# B&R Automation Studio project Panasonic_LinkaPowerCP2_A2021055 (part 14)

#### Variables.var - Local variables
```iecst
VAR
	FazaNavratu : UINT := 0;
	CasSrobovania : REAL := 0.0;
	PocetCisteniSkrutkovacky : USINT := 0;
	K30_PrevodMomentu : PrevodMomentu;
	M4_PrevodMomentu : PrevodMomentu;
	M5_PrevodMomentu : PrevodMomentu;
	CasEnable_1 : TON := (0);
	CasEnable_2 : TON;
	CasEnable_3 : TON;
	CasEnable_4 : TON;
	CasResetServo_1 : TON;
	CasResetServo_2 : TON;
	CasResetServo_3 : TON;
	CasResetServo_4 : TON;
	SC_SkrutkovaciSet_K30 : SequenceControlTyp := (0);
	SC_SkrutkovaciSet_M4 : SequenceControlTyp := (0);
	SC_SkrutkovaciSet_M5 : SequenceControlTyp := (0);
	TEST : BOOL := 0;
END_VAR
```

#### AtlasCopcoKomunikacia.st
```iecst
ACTION AtlasCopcoKomunikacia:

    M4_PrevodMomentu();
    M5_PrevodMomentu();
	K30_PrevodMomentu();
	//*********************************************************Skrutkovacka M5********************************************************************************//
	//Vstupy z AtlasCopco do PLC//
    P1_Srobovanie.Skrutkovacka_M5.Stav_VysledokPotvrdeny:= P1_Srobovanie.PAR.M5_AtlasCopcoInputs[0].0;
    P1_Srobovanie.Skrutkovacka_M5.Stav_EmergencyStop:= P1_Srobovanie.PAR.M5_AtlasCopcoInputs[0].1;
    P1_Srobovanie.Skrutkovacka_M5.Stav_READY_to_START:= P1_Srobovanie.PAR.M5_AtlasCopcoInputs[0].2;
    P1_Srobovanie.Skrutkovacka_M5.Stav_MANUAL:= P1_Srobovanie.PAR.M5_AtlasCopcoInputs[0].3;
    P1_Srobovanie.Skrutkovacka_M5.Stav_UtahovanieUkoncene:= P1_Srobovanie.PAR.M5_AtlasCopcoInputs[0].4;
    P1_Srobovanie.Skrutkovacka_M5.Stav_VysledokUtahovania_NG:= P1_Srobovanie.PAR.M5_AtlasCopcoInputs[0].5;
    P1_Srobovanie.Skrutkovacka_M5.Stav_VysledokUtahovania_OK:= P1_Srobovanie.PAR.M5_AtlasCopcoInputs[0].6;
    P1_Srobovanie.Skrutkovacka_M5.Stav_SmerOtacania_VPRED:= P1_Srobovanie.PAR.M5_AtlasCopcoInputs[0].7;
    P1_Srobovanie.Skrutkovacka_M5.Stav_BUSY:= P1_Srobovanie.PAR.M5_AtlasCopcoInputs[0].8;
    P1_Srobovanie.Skrutkovacka_M5.Stav_ControlerSwitch_ON:= P1_Srobovanie.PAR.M5_AtlasCopcoInputs[0].9;
    P1_Srobovanie.Skrutkovacka_M5.Stav_Station_READY:= P1_Srobovanie.PAR.M5_AtlasCopcoInputs[0].10;
    P1_Srobovanie.Skrutkovacka_M5.Stav_NastrojPripojeny:= P1_Srobovanie.PAR.M5_AtlasCopcoInputs[0].11;
    P1_Srobovanie.Skrutkovacka_M5.Stav_NastrojUtahuje:= P1_Srobovanie.PAR.M5_AtlasCopcoInputs[0].12;

    //Výstupy z PLC do AtlasCopco//
    P1_Srobovanie.PAR.M5_AtlasCopcoOutputs[0].0:= P1_Srobovanie.Skrutkovacka_M5.RESET_Poruchy;
    P1_Srobovanie.PAR.M5_AtlasCopcoOutputs[0].1:= P1_Srobovanie.Skrutkovacka_M5.RESET_Vysledkov;
    P1_Srobovanie.PAR.M5_AtlasCopcoOutputs[0].2:= P1_Srobovanie.Skrutkovacka_M5.START_Skrutkovania;
    P1_Srobovanie.PAR.M5_AtlasCopcoOutputs[0].3:= P1_Srobovanie.Skrutkovacka_M5.START_Utahovania;

    //Číslo zadaného programu//
    P1_Srobovanie.PAR.M5_AtlasCopcoOutputs[0].16:= P1_Srobovanie.Skrutkovacka_M5.CisloZadanehoProgramu.0;
    P1_Srobovanie.PAR.M5_AtlasCopcoOutputs[0].17:= P1_Srobovanie.Skrutkovacka_M5.CisloZadanehoProgramu.1;
    P1_Srobovanie.PAR.M5_AtlasCopcoOutputs[0].18:= P1_Srobovanie.Skrutkovacka_M5.CisloZadanehoProgramu.2;
    P1_Srobovanie.PAR.M5_AtlasCopcoOutputs[0].19:= P1_Srobovanie.Skrutkovacka_M5.CisloZadanehoProgramu.3;
    P1_Srobovanie.PAR.M5_AtlasCopcoOutputs[0].20:= P1_Srobovanie.Skrutkovacka_M5.CisloZadanehoProgramu.4;
    P1_Srobovanie.PAR.M5_AtlasCopcoOutputs[0].21:= P1_Srobovanie.Skrutkovacka_M5.CisloZadanehoProgramu.5;
    P1_Srobovanie.PAR.M5_AtlasCopcoOutputs[0].22:= P1_Srobovanie.Skrutkovacka_M5.CisloZadanehoProgramu.6;
    P1_Srobovanie.PAR.M5_AtlasCopcoOutputs[0].23:= P1_Srobovanie.Skrutkovacka_M5.CisloZadanehoProgramu.7;

    //Číslo aktuálneho programu//
    P1_Srobovanie.Skrutkovacka_M5.Stav_CisloAktualnehoProgramu.0:= P1_Srobovanie.PAR.M5_AtlasCopcoInputs[5].8;
    P1_Srobovanie.Skrutkovacka_M5.Stav_CisloAktualnehoProgramu.1:= P1_Srobovanie.PAR.M5_AtlasCopcoInputs[5].9;
    P1_Srobovanie.Skrutkovacka_M5.Stav_CisloAktualnehoProgramu.2:= P1_Srobovanie.PAR.M5_AtlasCopcoInputs[5].10;
    P1_Srobovanie.Skrutkovacka_M5.Stav_CisloAktualnehoProgramu.3:= P1_Srobovanie.PAR.M5_AtlasCopcoInputs[5].11;
    P1_Srobovanie.Skrutkovacka_M5.Stav_CisloAktualnehoProgramu.4:= P1_Srobovanie.PAR.M5_AtlasCopcoInputs[5].12;
    P1_Srobovanie.Skrutkovacka_M5.Stav_CisloAktualnehoProgramu.5:= P1_Srobovanie.PAR.M5_AtlasCopcoInputs[5].13;
    P1_Srobovanie.Skrutkovacka_M5.Stav_CisloAktualnehoProgramu.6:= P1_Srobovanie.PAR.M5_AtlasCopcoInputs[5].14;
    P1_Srobovanie.Skrutkovacka_M5.Stav_CisloAktualnehoProgramu.7:= P1_Srobovanie.PAR.M5_AtlasCopcoInputs[5].15;

    //Program č.1 - skrutkovanie do plastu
    //Program č.2 - skrutkovanie do kovu

    //Dosiahnutý moment//
//    P1_Srobovanie.STAV.M5_DosiahnutyMoment.0:= P1_Srobovanie.PAR.M5_AtlasCopcoInputs[1].24;
//    P1_Srobovanie.STAV.M5_DosiahnutyMoment.1:= P1_Srobovanie.PAR.M5_AtlasCopcoInputs[1].25;
//    P1_Srobovanie.STAV.M5_DosiahnutyMoment.2:= P1_Srobovanie.PAR.M5_AtlasCopcoInputs[1].26;
//    P1_Srobovanie.STAV.M5_DosiahnutyMoment.3:= P1_Srobovanie.PAR.M5_AtlasCopcoInputs[1].27;
//    P1_Srobovanie.STAV.M5_DosiahnutyMoment.4:= P1_Srobovanie.PAR.M5_AtlasCopcoInputs[1].28;
//    P1_Srobovanie.STAV.M5_DosiahnutyMoment.5:= P1_Srobovanie.PAR.M5_AtlasCopcoInputs[1].29;
//    P1_Srobovanie.STAV.M5_DosiahnutyMoment.6:= P1_Srobovanie.PAR.M5_AtlasCopcoInputs[1].30;
//    P1_Srobovanie.STAV.M5_DosiahnutyMoment.7:= P1_Srobovanie.PAR.M5_AtlasCopcoInputs[1].31;
//    P1_Srobovanie.STAV.M5_DosiahnutyMoment.8:= P1_Srobovanie.PAR.M5_AtlasCopcoInputs[1].16;
//    P1_Srobovanie.STAV.M5_DosiahnutyMoment.9:= P1_Srobovanie.PAR.M5_AtlasCopcoInputs[1].17;
//    P1_Srobovanie.STAV.M5_DosiahnutyMoment.10:= P1_Srobovanie.PAR.M5_AtlasCopcoInputs[1].18;
//    P1_Srobovanie.STAV.M5_DosiahnutyMoment.11:= P1_Srobovanie.PAR.M5_AtlasCopcoInputs[1].19;
//    P1_Srobovanie.STAV.M5_DosiahnutyMoment.12:= P1_Srobovanie.PAR.M5_AtlasCopcoInputs[1].20;
//    P1_Srobovanie.STAV.M5_DosiahnutyMoment.13:= P1_Srobovanie.PAR.M5_AtlasCopcoInputs[1].21;
//    P1_Srobovanie.STAV.M5_DosiahnutyMoment.14:= P1_Srobovanie.PAR.M5_AtlasCopcoInputs[1].22;
//    P1_Srobovanie.STAV.M5_DosiahnutyMoment.15:= P1_Srobovanie.PAR.M5_AtlasCopcoInputs[1].23;
//    P1_Srobovanie.STAV.M5_DosiahnutyMoment.16:= P1_Srobovanie.PAR.M5_AtlasCopcoInputs[1].8;
//    P1_Srobovanie.STAV.M5_DosiahnutyMoment.17:= P1_Srobovanie.PAR.M5_AtlasCopcoInputs[1].9;
//    P1_Srobovanie.STAV.M5_DosiahnutyMoment.18:= P1_Srobovanie.PAR.M5_AtlasCopcoInputs[1].10;
//    P1_Srobovanie.STAV.M5_DosiahnutyMoment.19:= P1_Srobovanie.PAR.M5_AtlasCopcoInputs[1].11;
//    P1_Srobovanie.STAV.M5_DosiahnutyMoment.20:= P1_Srobovanie.PAR.M5_AtlasCopcoInputs[1].12;
//    P1_Srobovanie.STAV.M5_DosiahnutyMoment.21:= P1_Srobovanie.PAR.M5_AtlasCopcoInputs[1].13;
//    P1_Srobovanie.STAV.M5_DosiahnutyMoment.22:= P1_Srobovanie.PAR.M5_AtlasCopcoInputs[1].14;
//    P1_Srobovanie.STAV.M5_DosiahnutyMoment.23:= P1_Srobovanie.PAR.M5_AtlasCopcoInputs[1].15;
//    P1_Srobovanie.STAV.M5_DosiahnutyMoment.24:= P1_Srobovanie.PAR.M5_AtlasCopcoInputs[1].0;
//    P1_Srobovanie.STAV.M5_DosiahnutyMoment.25:= P1_Srobovanie.PAR.M5_AtlasCopcoInputs[1].1;
//    P1_Srobovanie.STAV.M5_DosiahnutyMoment.26:= P1_Srobovanie.PAR.M5_AtlasCopcoInputs[1].2;
//    P1_Srobovanie.STAV.M5_DosiahnutyMoment.27:= P1_Srobovanie.PAR.M5_AtlasCopcoInputs[1].3;
//    P1_Srobovanie.STAV.M5_DosiahnutyMoment.28:= P1_Srobovanie.PAR.M5_AtlasCopcoInputs[1].4;
//    P1_Srobovanie.STAV.M5_DosiahnutyMoment.29:= P1_Srobovanie.PAR.M5_AtlasCopcoInputs[1].5;
//    P1_Srobovanie.STAV.M5_DosiahnutyMoment.30:= P1_Srobovanie.PAR.M5_AtlasCopcoInputs[1].6;
//    P1_Srobovanie.STAV.M5_DosiahnutyMoment.31:= P1_Srobovanie.PAR.M5_AtlasCopcoInputs[1].7;
//    M5_DosiahnutyMoment_REAL:= UDINT_TO_REAL(P1_Srobovanie.STAV.M5_DosiahnutyMoment);
//    IF M5_DosiahnutyMoment_REAL > 0 THEN
//        P1_Srobovanie.STAV.M5_DosiahnutyMoment_REAL:= M5_DosiahnutyMoment_REAL/100;
//    ELSE
//        P1_Srobovanie.STAV.M5_DosiahnutyMoment_REAL:= 0.0;
//    END_IF

    M5_PrevodMomentu.AtlasAktualnyMoment:=P1_Srobovanie.PAR.M5_AtlasCopcoInputs[1];
    P1_Srobovanie.STAV.M5_DosiahnutyMoment_REAL:=M5_PrevodMomentu.AktualnyMoment;

    //Moment - Tolerancia MAX//
//    P1_Srobovanie.STAV.M5_Moment_ToleranciaMAX.0:= P1_Srobovanie.PAR.M5_AtlasCopcoInputs[3].24;
//    P1_Srobovanie.STAV.M5_Moment_ToleranciaMAX.1:= P1_Srobovanie.PAR.M5_AtlasCopcoInputs[3].25;
//    P1_Srobovanie.STAV.M5_Moment_ToleranciaMAX.2:= P1_Srobovanie.PAR.M5_AtlasCopcoInputs[3].26;
//    P1_Srobovanie.STAV.M5_Moment_ToleranciaMAX.3:= P1_Srobovanie.PAR.M5_AtlasCopcoInputs[3].27;
//    P1_Srobovanie.STAV.M5_Moment_ToleranciaMAX.4:= P1_Srobovanie.PAR.M5_AtlasCopcoInputs[3].28;
//    P1_Srobovanie.STAV.M5_Moment_ToleranciaMAX.5:= P1_Srobovanie.PAR.M5_AtlasCopcoInputs[3].29;
//    P1_Srobovanie.STAV.M5_Moment_ToleranciaMAX.6:= P1_Srobovanie.PAR.M5_AtlasCopcoInputs[3].30;
//    P1_Srobovanie.STAV.M5_Moment_ToleranciaMAX.7:= P1_Srobovanie.PAR.M5_AtlasCopcoInputs[3].31;
//    P1_Srobovanie.STAV.M5_Moment_ToleranciaMAX.8:= P1_Srobovanie.PAR.M5_AtlasCopcoInputs[3].16;
//    P1_Srobovanie.STAV.M5_Moment_ToleranciaMAX.9:= P1_Srobovanie.PAR.M5_AtlasCopcoInputs[3].17;
//    P1_Srobovanie.STAV.M5_Moment_ToleranciaMAX.10:= P1_Srobovanie.PAR.M5_AtlasCopcoInputs[3].18;
//    P1_Srobovanie.STAV.M5_Moment_ToleranciaMAX.11:= P1_Srobovanie.PAR.M5_AtlasCopcoInputs[3].19;
//    P1_Srobovanie.STAV.M5_Moment_ToleranciaMAX.12:= P1_Srobovanie.PAR.M5_AtlasCopcoInputs[3].20;
//    P1_Srobovanie.STAV.M5_Moment_ToleranciaMAX.13:= P1_Srobovanie.PAR.M5_AtlasCopcoInputs[3].21;
//    P1_Srobovanie.STAV.M5_Moment_ToleranciaMAX.14:= P1_Srobovanie.PAR.M5_AtlasCopcoInputs[3].22;
//    P1_Srobovanie.STAV.M5_Moment_ToleranciaMAX.15:= P1_Srobovanie.PAR.M5_AtlasCopcoInputs[3].23;
//    P1_Srobovanie.STAV.M5_Moment_ToleranciaMAX.16:= P1_Srobovanie.PAR.M5_AtlasCopcoInputs[3].8;
//    P1_Srobovanie.STAV.M5_Moment_ToleranciaMAX.17:= P1_Srobovanie.PAR.M5_AtlasCopcoInputs[3].9;
//    P1_Srobovanie.STAV.M5_Moment_ToleranciaMAX.18:= P1_Srobovanie.PAR.M5_AtlasCopcoInputs[3].10;
//    P1_Srobovanie.STAV.M5_Moment_ToleranciaMAX.19:= P1_Srobovanie.PAR.M5_AtlasCopcoInputs[3].11;
//    P1_Srobovanie.STAV.M5_Moment_ToleranciaMAX.20:= P1_Srobovanie.PAR.M5_AtlasCopcoInputs[3].12;
//    P1_Srobovanie.STAV.M5_Moment_ToleranciaMAX.21:= P1_Srobovanie.PAR.M5_AtlasCopcoInputs[3].13;
//    P1_Srobovanie.STAV.M5_Moment_ToleranciaMAX.22:= P1_Srobovanie.PAR.M5_AtlasCopcoInputs[3].14;
//    P1_Srobovanie.STAV.M5_Moment_ToleranciaMAX.23:= P1_Srobovanie.PAR.M5_AtlasCopcoInputs[3].15;
//    P1_Srobovanie.STAV.M5_Moment_ToleranciaMAX.24:= P1_Srobovanie.PAR.M5_AtlasCopcoInputs[3].0;
//    P1_Srobovanie.STAV.M5_Moment_ToleranciaMAX.25:= P1_Srobovanie.PAR.M5_AtlasCopcoInputs[3].1;
//    P1_Srobovanie.STAV.M5_Moment_ToleranciaMAX.26:= P1_Srobovanie.PAR.M5_AtlasCopcoInputs[3].2;
//    P1_Srobovanie.STAV.M5_Moment_ToleranciaMAX.27:= P1_Srobovanie.PAR.M5_AtlasCopcoInputs[3].3;
//    P1_Srobovanie.STAV.M5_Moment_ToleranciaMAX.28:= P1_Srobovanie.PAR.M5_AtlasCopcoInputs[3].4;
//    P1_Srobovanie.STAV.M5_Moment_ToleranciaMAX.29:= P1_Srobovanie.PAR.M5_AtlasCopcoInputs[3].5;
//    P1_Srobovanie.STAV.M5_Moment_ToleranciaMAX.30:= P1_Srobovanie.PAR.M5_AtlasCopcoInputs[3].6;
//    P1_Srobovanie.STAV.M5_Moment_ToleranciaMAX.31:= P1_Srobovanie.PAR.M5_AtlasCopcoInputs[3].7;
//    M5_Moment_ToleranciaMAX_REAL:= UDINT_TO_REAL(P1_Srobovanie.STAV.M5_Moment_ToleranciaMAX);
//    IF M5_Moment_ToleranciaMAX_REAL > 0 THEN
//        P1_Srobovanie.STAV.M5_Moment_ToleranciaMAX_REAL:= M5_Moment_ToleranciaMAX_REAL/100;
//    ELSE
//        P1_Srobovanie.STAV.M5_Moment_ToleranciaMAX_REAL:= 0.0;
    //    END_IF

    M5_PrevodMomentu.AtlasMaximalnaTolerancia:=P1_Srobovanie.PAR.M5_AtlasCopcoInputs[3];
    P1_Srobovanie.STAV.M5_Moment_ToleranciaMAX_REAL:=M5_PrevodMomentu.ToleranciaMAX;

    //Moment - Tolerancia MIN//
//    P1_Srobovanie.STAV.M5_Moment_ToleranciaMIN.0:= P1_Srobovanie.PAR.M5_AtlasCopcoInputs[4].24;
//    P1_Srobovanie.STAV.M5_Moment_ToleranciaMIN.1:= P1_Srobovanie.PAR.M5_AtlasCopcoInputs[4].25;
//    P1_Srobovanie.STAV.M5_Moment_ToleranciaMIN.2:= P1_Srobovanie.PAR.M5_AtlasCopcoInputs[4].26;
//    P1_Srobovanie.STAV.M5_Moment_ToleranciaMIN.3:= P1_Srobovanie.PAR.M5_AtlasCopcoInputs[4].27;
//    P1_Srobovanie.STAV.M5_Moment_ToleranciaMIN.4:= P1_Srobovanie.PAR.M5_AtlasCopcoInputs[4].28;
//    P1_Srobovanie.STAV.M5_Moment_ToleranciaMIN.5:= P1_Srobovanie.PAR.M5_AtlasCopcoInputs[4].29;
//    P1_Srobovanie.STAV.M5_Moment_ToleranciaMIN.6:= P1_Srobovanie.PAR.M5_AtlasCopcoInputs[4].30;
//    P1_Srobovanie.STAV.M5_Moment_ToleranciaMIN.7:= P1_Srobovanie.PAR.M5_AtlasCopcoInputs[4].31;
//    P1_Srobovanie.STAV.M5_Moment_ToleranciaMIN.8:= P1_Srobovanie.PAR.M5_AtlasCopcoInputs[4].16;
//    P1_Srobovanie.STAV.M5_Moment_ToleranciaMIN.9:= P1_Srobovanie.PAR.M5_AtlasCopcoInputs[4].17;
//    P1_Srobovanie.STAV.M5_Moment_ToleranciaMIN.10:= P1_Srobovanie.PAR.M5_AtlasCopcoInputs[4].18;
//    P1_Srobovanie.STAV.M5_Moment_ToleranciaMIN.11:= P1_Srobovanie.PAR.M5_AtlasCopcoInputs[4].19;
//    P1_Srobovanie.STAV.M5_Moment_ToleranciaMIN.12:= P1_Srobovanie.PAR.M5_AtlasCopcoInputs[4].20;
//    P1_Srobovanie.STAV.M5_Moment_ToleranciaMIN.13:= P1_Srobovanie.PAR.M5_AtlasCopcoInputs[4].21;
//    P1_Srobovanie.STAV.M5_Moment_ToleranciaMIN.14:= P1_Srobovanie.PAR.M5_AtlasCopcoInputs[4].22;
//    P1_Srobovanie.STAV.M5_Moment_ToleranciaMIN.15:= P1_Srobovanie.PAR.M5_AtlasCopcoInputs[4].23;
//    P1_Srobovanie.STAV.M5_Moment_ToleranciaMIN.16:= P1_Srobovanie.PAR.M5_AtlasCopcoInputs[4].8;
//    P1_Srobovanie.STAV.M5_Moment_ToleranciaMIN.17:= P1_Srobovanie.PAR.M5_AtlasCopcoInputs[4].9;
//    P1_Srobovanie.STAV.M5_Moment_ToleranciaMIN.18:= P1_Srobovanie.PAR.M5_AtlasCopcoInputs[4].10;
//    P1_Srobovanie.STAV.M5_Moment_ToleranciaMIN.19:= P1_Srobovanie.PAR.M5_AtlasCopcoInputs[4].11;
//    P1_Srobovanie.STAV.M5_Moment_ToleranciaMIN.20:= P1_Srobovanie.PAR.M5_AtlasCopcoInputs[4].12;
//    P1_Srobovanie.STAV.M5_Moment_ToleranciaMIN.21:= P1_Srobovanie.PAR.M5_AtlasCopcoInputs[4].13;
//    P1_Srobovanie.STAV.M5_Moment_ToleranciaMIN.22:= P1_Srobovanie.PAR.M5_AtlasCopcoInputs[4].14;
//    P1_Srobovanie.STAV.M5_Moment_ToleranciaMIN.23:= P1_Srobovanie.PAR.M5_AtlasCopcoInputs[4].15;
//    P1_Srobovanie.STAV.M5_Moment_ToleranciaMIN.24:= P1_Srobovanie.PAR.M5_AtlasCopcoInputs[4].0;
//    P1_Srobovanie.STAV.M5_Moment_ToleranciaMIN.25:= P1_Srobovanie.PAR.M5_AtlasCopcoInputs[4].1;
//    P1_Srobovanie.STAV.M5_Moment_ToleranciaMIN.26:= P1_Srobovanie.PAR.M5_AtlasCopcoInputs[4].2;
//    P1_Srobovanie.STAV.M5_Moment_ToleranciaMIN.27:= P1_Srobovanie.PAR.M5_AtlasCopcoInputs[4].3;
//    P1_Srobovanie.STAV.M5_Moment_ToleranciaMIN.28:= P1_Srobovanie.PAR.M5_AtlasCopcoInputs[4].4;
//    P1_Srobovanie.STAV.M5_Moment_ToleranciaMIN.29:= P1_Srobovanie.PAR.M5_AtlasCopcoInputs[4].5;
//    P1_Srobovanie.STAV.M5_Moment_ToleranciaMIN.30:= P1_Srobovanie.PAR.M5_AtlasCopcoInputs[4].6;
//    P1_Srobovanie.STAV.M5_Moment_ToleranciaMIN.31:= P1_Srobovanie.PAR.M5_AtlasCopcoInputs[4].7;
//    M5_Moment_ToleranciaMIN_REAL:= UDINT_TO_REAL(P1_Srobovanie.STAV.M5_Moment_ToleranciaMIN);
//    IF M5_Moment_ToleranciaMIN_REAL > 0 THEN
//        P1_Srobovanie.STAV.M5_Moment_ToleranciaMIN_REAL:= M5_Moment_ToleranciaMIN_REAL /100;
//    ELSE
//        P1_Srobovanie.STAV.M5_Moment_ToleranciaMIN_REAL:= 0.0;
    //    END_IF

    M5_PrevodMomentu.AtlasMinimalnaTolerancia:=P1_Srobovanie.PAR.M5_AtlasCopcoInputs[4];
    P1_Srobovanie.STAV.M5_Moment_ToleranciaMIN_REAL:=M5_PrevodMomentu.ToleranciaMIN;

    //Dosiahnutý úhol//
    P1_Srobovanie.STAV.M5_DosiahnutyUhol.0:= P1_Srobovanie.PAR.M5_AtlasCopcoInputs[0].24;
    P1_Srobovanie.STAV.M5_DosiahnutyUhol.1:= P1_Srobovanie.PAR.M5_AtlasCopcoInputs[0].25;
    P1_Srobovanie.STAV.M5_DosiahnutyUhol.2:= P1_Srobovanie.PAR.M5_AtlasCopcoInputs[0].26;
    P1_Srobovanie.STAV.M5_DosiahnutyUhol.3:= P1_Srobovanie.PAR.M5_AtlasCopcoInputs[0].27;
    P1_Srobovanie.STAV.M5_DosiahnutyUhol.4:= P1_Srobovanie.PAR.M5_AtlasCopcoInputs[0].28;
    P1_Srobovanie.STAV.M5_DosiahnutyUhol.5:= P1_Srobovanie.PAR.M5_AtlasCopcoInputs[0].29;
    P1_Srobovanie.STAV.M5_DosiahnutyUhol.6:= P1_Srobovanie.PAR.M5_AtlasCopcoInputs[0].30;
    P1_Srobovanie.STAV.M5_DosiahnutyUhol.7:= P1_Srobovanie.PAR.M5_AtlasCopcoInputs[0].31;
    P1_Srobovanie.STAV.M5_DosiahnutyUhol.8:= P1_Srobovanie.PAR.M5_AtlasCopcoInputs[0].16;
    P1_Srobovanie.STAV.M5_DosiahnutyUhol.9:= P1_Srobovanie.PAR.M5_AtlasCopcoInputs[0].17;
    P1_Srobovanie.STAV.M5_DosiahnutyUhol.10:= P1_Srobovanie.PAR.M5_AtlasCopcoInputs[0].18;
    P1_Srobovanie.STAV.M5_DosiahnutyUhol.11:= P1_Srobovanie.PAR.M5_AtlasCopcoInputs[0].19;
    P1_Srobovanie.STAV.M5_DosiahnutyUhol.12:= P1_Srobovanie.PAR.M5_AtlasCopcoInputs[0].20;
    P1_Srobovanie.STAV.M5_DosiahnutyUhol.13:= P1_Srobovanie.PAR.M5_AtlasCopcoInputs[0].21;
    P1_Srobovanie.STAV.M5_DosiahnutyUhol.14:= P1_Srobovanie.PAR.M5_AtlasCopcoInputs[0].22;
    P1_Srobovanie.STAV.M5_DosiahnutyUhol.15:= P1_Srobovanie.PAR.M5_AtlasCopcoInputs[0].23;

    //Uhol - Tolerancia MAX//
    P1_Srobovanie.STAV.M5_Uhol_ToleranciaMAX.0:= P1_Srobovanie.PAR.M5_AtlasCopcoInputs[2].8;
    P1_Srobovanie.STAV.M5_Uhol_ToleranciaMAX.1:= P1_Srobovanie.PAR.M5_AtlasCopcoInputs[2].9;
    P1_Srobovanie.STAV.M5_Uhol_ToleranciaMAX.2:= P1_Srobovanie.PAR.M5_AtlasCopcoInputs[2].10;
    P1_Srobovanie.STAV.M5_Uhol_ToleranciaMAX.3:= P1_Srobovanie.PAR.M5_AtlasCopcoInputs[2].11;
    P1_Srobovanie.STAV.M5_Uhol_ToleranciaMAX.4:= P1_Srobovanie.PAR.M5_AtlasCopcoInputs[2].12;
    P1_Srobovanie.STAV.M5_Uhol_ToleranciaMAX.5:= P1_Srobovanie.PAR.M5_AtlasCopcoInputs[2].13;
    P1_Srobovanie.STAV.M5_Uhol_ToleranciaMAX.6:= P1_Srobovanie.PAR.M5_AtlasCopcoInputs[2].14;
    P1_Srobovanie.STAV.M5_Uhol_ToleranciaMAX.7:= P1_Srobovanie.PAR.M5_AtlasCopcoInputs[2].15;
    P1_Srobovanie.STAV.M5_Uhol_ToleranciaMAX.8:= P1_Srobovanie.PAR.M5_AtlasCopcoInputs[2].0;
    P1_Srobovanie.STAV.M5_Uhol_ToleranciaMAX.9:= P1_Srobovanie.PAR.M5_AtlasCopcoInputs[2].1;
    P1_Srobovanie.STAV.M5_Uhol_ToleranciaMAX.10:= P1_Srobovanie.PAR.M5_AtlasCopcoInputs[2].2;
    P1_Srobovanie.STAV.M5_Uhol_ToleranciaMAX.11:= P1_Srobovanie.PAR.M5_AtlasCopcoInputs[2].3;
    P1_Srobovanie.STAV.M5_Uhol_ToleranciaMAX.12:= P1_Srobovanie.PAR.M5_AtlasCopcoInputs[2].4;
    P1_Srobovanie.STAV.M5_Uhol_ToleranciaMAX.13:= P1_Srobovanie.PAR.M5_AtlasCopcoInputs[2].5;
    P1_Srobovanie.STAV.M5_Uhol_ToleranciaMAX.14:= P1_Srobovanie.PAR.M5_AtlasCopcoInputs[2].6;
    P1_Srobovanie.STAV.M5_Uhol_ToleranciaMAX.15:= P1_Srobovanie.PAR.M5_AtlasCopcoInputs[2].7;

    //Uhol - Tolerancia MIN//
    P1_Srobovanie.STAV.M5_Uhol_ToleranciaMIN.0:= P1_Srobovanie.PAR.M5_AtlasCopcoInputs[2].24;
    P1_Srobovanie.STAV.M5_Uhol_ToleranciaMIN.1:= P1_Srobovanie.PAR.M5_AtlasCopcoInputs[2].25;
    P1_Srobovanie.STAV.M5_Uhol_ToleranciaMIN.2:= P1_Srobovanie.PAR.M5_AtlasCopcoInputs[2].26;
    P1_Srobovanie.STAV.M5_Uhol_ToleranciaMIN.3:= P1_Srobovanie.PAR.M5_AtlasCopcoInputs[2].27;
    P1_Srobovanie.STAV.M5_Uhol_ToleranciaMIN.4:= P1_Srobovanie.PAR.M5_AtlasCopcoInputs[2].28;
    P1_Srobovanie.STAV.M5_Uhol_ToleranciaMIN.5:= P1_Srobovanie.PAR.M5_AtlasCopcoInputs[2].29;
    P1_Srobovanie.STAV.M5_Uhol_ToleranciaMIN.6:= P1_Srobovanie.PAR.M5_AtlasCopcoInputs[2].30;
    P1_Srobovanie.STAV.M5_Uhol_ToleranciaMIN.7:= P1_Srobovanie.PAR.M5_AtlasCopcoInputs[2].31;
    P1_Srobovanie.STAV.M5_Uhol_ToleranciaMIN.8:= P1_Srobovanie.PAR.M5_AtlasCopcoInputs[2].16;
    P1_Srobovanie.STAV.M5_Uhol_ToleranciaMIN.9:= P1_Srobovanie.PAR.M5_AtlasCopcoInputs[2].17;
    P1_Srobovanie.STAV.M5_Uhol_ToleranciaMIN.10:= P1_Srobovanie.PAR.M5_AtlasCopcoInputs[2].18;
    P1_Srobovanie.STAV.M5_Uhol_ToleranciaMIN.11:= P1_Srobovanie.PAR.M5_AtlasCopcoInputs[2].19;
    P1_Srobovanie.STAV.M5_Uhol_ToleranciaMIN.12:= P1_Srobovanie.PAR.M5_AtlasCopcoInputs[2].20;
    P1_Srobovanie.STAV.M5_Uhol_ToleranciaMIN.13:= P1_Srobovanie.PAR.M5_AtlasCopcoInputs[2].21;
    P1_Srobovanie.STAV.M5_Uhol_ToleranciaMIN.14:= P1_Srobovanie.PAR.M5_AtlasCopcoInputs[2].22;
    P1_Srobovanie.STAV.M5_Uhol_ToleranciaMIN.15:= P1_Srobovanie.PAR.M5_AtlasCopcoInputs[2].23;

    //***************************************************************Skrutkovacka M4************************************************************************************//
    //Vstupy z AtlasCopco do PLC//
    P1_Srobovanie.Skrutkovacka_M4.Stav_VysledokPotvrdeny:= P1_Srobovanie.PAR.M4_AtlasCopcoInputs[0].0;
    P1_Srobovanie.Skrutkovacka_M4.Stav_EmergencyStop:= P1_Srobovanie.PAR.M4_AtlasCopcoInputs[0].1;
    P1_Srobovanie.Skrutkovacka_M4.Stav_READY_to_START:= P1_Srobovanie.PAR.M4_AtlasCopcoInputs[0].2;
    P1_Srobovanie.Skrutkovacka_M4.Stav_MANUAL:= P1_Srobovanie.PAR.M4_AtlasCopcoInputs[0].3;
    P1_Srobovanie.Skrutkovacka_M4.Stav_UtahovanieUkoncene:= P1_Srobovanie.PAR.M4_AtlasCopcoInputs[0].4;
    P1_Srobovanie.Skrutkovacka_M4.Stav_VysledokUtahovania_NG:= P1_Srobovanie.PAR.M4_AtlasCopcoInputs[0].5;
    P1_Srobovanie.Skrutkovacka_M4.Stav_VysledokUtahovania_OK:= P1_Srobovanie.PAR.M4_AtlasCopcoInputs[0].6;
    P1_Srobovanie.Skrutkovacka_M4.Stav_SmerOtacania_VPRED:= P1_Srobovanie.PAR.M4_AtlasCopcoInputs[0].7;
    P1_Srobovanie.Skrutkovacka_M4.Stav_BUSY:= P1_Srobovanie.PAR.M4_AtlasCopcoInputs[0].8;
    P1_Srobovanie.Skrutkovacka_M4.Stav_ControlerSwitch_ON:= P1_Srobovanie.PAR.M4_AtlasCopcoInputs[0].9;
    P1_Srobovanie.Skrutkovacka_M4.Stav_Station_READY:= P1_Srobovanie.PAR.M4_AtlasCopcoInputs[0].10;
    P1_Srobovanie.Skrutkovacka_M4.Stav_NastrojPripojeny:= P1_Srobovanie.PAR.M4_AtlasCopcoInputs[0].11;
    P1_Srobovanie.Skrutkovacka_M4.Stav_NastrojUtahuje:= P1_Srobovanie.PAR.M4_AtlasCopcoInputs[0].12;

    //Výstupy z PLC do AtlasCopco//
    P1_Srobovanie.PAR.M4_AtlasCopcoOutputs[0].0:= P1_Srobovanie.Skrutkovacka_M4.RESET_Poruchy;
    P1_Srobovanie.PAR.M4_AtlasCopcoOutputs[0].1:= P1_Srobovanie.Skrutkovacka_M4.RESET_Vysledkov;
    P1_Srobovanie.PAR.M4_AtlasCopcoOutputs[0].2:= P1_Srobovanie.Skrutkovacka_M4.START_Skrutkovania;
    P1_Srobovanie.PAR.M4_AtlasCopcoOutputs[0].3:= P1_Srobovanie.Skrutkovacka_M4.START_Utahovania;

    //Dosiahnutý moment//
//    P1_Srobovanie.STAV.M4_DosiahnutyMoment.0:= P1_Srobovanie.PAR.M4_AtlasCopcoInputs[1].24;
//    P1_Srobovanie.STAV.M4_DosiahnutyMoment.1:= P1_Srobovanie.PAR.M4_AtlasCopcoInputs[1].25;
//    P1_Srobovanie.STAV.M4_DosiahnutyMoment.2:= P1_Srobovanie.PAR.M4_AtlasCopcoInputs[1].26;
//    P1_Srobovanie.STAV.M4_DosiahnutyMoment.3:= P1_Srobovanie.PAR.M4_AtlasCopcoInputs[1].27;
//    P1_Srobovanie.STAV.M4_DosiahnutyMoment.4:= P1_Srobovanie.PAR.M4_AtlasCopcoInputs[1].28;
//    P1_Srobovanie.STAV.M4_DosiahnutyMoment.5:= P1_Srobovanie.PAR.M4_AtlasCopcoInputs[1].29;
//    P1_Srobovanie.STAV.M4_DosiahnutyMoment.6:= P1_Srobovanie.PAR.M4_AtlasCopcoInputs[1].30;
//    P1_Srobovanie.STAV.M4_DosiahnutyMoment.7:= P1_Srobovanie.PAR.M4_AtlasCopcoInputs[1].31;
//    P1_Srobovanie.STAV.M4_DosiahnutyMoment.8:= P1_Srobovanie.PAR.M4_AtlasCopcoInputs[1].16;
//    P1_Srobovanie.STAV.M4_DosiahnutyMoment.9:= P1_Srobovanie.PAR.M4_AtlasCopcoInputs[1].17;
//    P1_Srobovanie.STAV.M4_DosiahnutyMoment.10:= P1_Srobovanie.PAR.M4_AtlasCopcoInputs[1].18;
//    P1_Srobovanie.STAV.M4_DosiahnutyMoment.11:= P1_Srobovanie.PAR.M4_AtlasCopcoInputs[1].19;
//    P1_Srobovanie.STAV.M4_DosiahnutyMoment.12:= P1_Srobovanie.PAR.M4_AtlasCopcoInputs[1].20;
//    P1_Srobovanie.STAV.M4_DosiahnutyMoment.13:= P1_Srobovanie.PAR.M4_AtlasCopcoInputs[1].21;
//    P1_Srobovanie.STAV.M4_DosiahnutyMoment.14:= P1_Srobovanie.PAR.M4_AtlasCopcoInputs[1].22;
//    P1_Srobovanie.STAV.M4_DosiahnutyMoment.15:= P1_Srobovanie.PAR.M4_AtlasCopcoInputs[1].23;
//    P1_Srobovanie.STAV.M4_DosiahnutyMoment.16:= P1_Srobovanie.PAR.M4_AtlasCopcoInputs[1].8;
//    P1_Srobovanie.STAV.M4_DosiahnutyMoment.17:= P1_Srobovanie.PAR.M4_AtlasCopcoInputs[1].9;
//    P1_Srobovanie.STAV.M4_DosiahnutyMoment.18:= P1_Srobovanie.PAR.M4_AtlasCopcoInputs[1].10;
//    P1_Srobovanie.STAV.M4_DosiahnutyMoment.19:= P1_Srobovanie.PAR.M4_AtlasCopcoInputs[1].11;
//    P1_Srobovanie.STAV.M4_DosiahnutyMoment.20:= P1_Srobovanie.PAR.M4_AtlasCopcoInputs[1].12;
//    P1_Srobovanie.STAV.M4_DosiahnutyMoment.21:= P1_Srobovanie.PAR.M4_AtlasCopcoInputs[1].13;
//    P1_Srobovanie.STAV.M4_DosiahnutyMoment.22:= P1_Srobovanie.PAR.M4_AtlasCopcoInputs[1].14;
//    P1_Srobovanie.STAV.M4_DosiahnutyMoment.23:= P1_Srobovanie.PAR.M4_AtlasCopcoInputs[1].15;
//    P1_Srobovanie.STAV.M4_DosiahnutyMoment.24:= P1_Srobovanie.PAR.M4_AtlasCopcoInputs[1].0;
//    P1_Srobovanie.STAV.M4_DosiahnutyMoment.25:= P1_Srobovanie.PAR.M4_AtlasCopcoInputs[1].1;
//    P1_Srobovanie.STAV.M4_DosiahnutyMoment.26:= P1_Srobovanie.PAR.M4_AtlasCopcoInputs[1].2;
//    P1_Srobovanie.STAV.M4_DosiahnutyMoment.27:= P1_Srobovanie.PAR.M4_AtlasCopcoInputs[1].3;
//    P1_Srobovanie.STAV.M4_DosiahnutyMoment.28:= P1_Srobovanie.PAR.M4_AtlasCopcoInputs[1].4;
//    P1_Srobovanie.STAV.M4_DosiahnutyMoment.29:= P1_Srobovanie.PAR.M4_AtlasCopcoInputs[1].5;
//    P1_Srobovanie.STAV.M4_DosiahnutyMoment.30:= P1_Srobovanie.PAR.M4_AtlasCopcoInputs[1].6;
//    P1_Srobovanie.STAV.M4_DosiahnutyMoment.31:= P1_Srobovanie.PAR.M4_AtlasCopcoInputs[1].7;
//    M4_DosiahnutyMoment_REAL:= UDINT_TO_REAL(P1_Srobovanie.STAV.M4_DosiahnutyMoment);
//    IF M4_DosiahnutyMoment_REAL > 0 THEN
//        P1_Srobovanie.STAV.M4_DosiahnutyMoment_REAL:= (M4_DosiahnutyMoment_REAL*0.65)/42598;
//    ELSE
//        P1_Srobovanie.STAV.M4_DosiahnutyMoment_REAL:= 0.0;
//    END_IF

    M4_PrevodMomentu.AtlasAktualnyMoment:=P1_Srobovanie.PAR.M4_AtlasCopcoInputs[1];
    P1_Srobovanie.STAV.M4_DosiahnutyMoment_REAL:=M4_PrevodMomentu.AktualnyMoment;

    (*P1_Srobovanie.STAV.M4_DosiahnutyMoment_REAL:= M4_DosiahnutyMoment_REAL/100;*)

    //Moment - Tolerancia MAX//
//    P1_Srobovanie.STAV.M4_Moment_ToleranciaMAX.0:= P1_Srobovanie.PAR.M4_AtlasCopcoInputs[3].24;
    //    P1_Srobovanie.STAV.M4_Moment_ToleranciaMAX.1:= P1_Srobovanie.PAR.M4_AtlasCopcoInputs[3].25;
//    P1_Srobovanie.STAV.M4_Moment_ToleranciaMAX.2:= P1_Srobovanie.PAR.M4_AtlasCopcoInputs[3].26;
//    P1_Srobovanie.STAV.M4_Moment_ToleranciaMAX.3:= P1_Srobovanie.PAR.M4_AtlasCopcoInputs[3].27;
//    P1_Srobovanie.STAV.M4_Moment_ToleranciaMAX.4:= P1_Srobovanie.PAR.M4_AtlasCopcoInputs[3].28;
//    P1_Srobovanie.STAV.M4_Moment_ToleranciaMAX.5:= P1_Srobovanie.PAR.M4_AtlasCopcoInputs[3].29;
//    P1_Srobovanie.STAV.M4_Moment_ToleranciaMAX.6:= P1_Srobovanie.PAR.M4_AtlasCopcoInputs[3].30;
//    P1_Srobovanie.STAV.M4_Moment_ToleranciaMAX.7:= P1_Srobovanie.PAR.M4_AtlasCopcoInputs[3].31;
//    P1_Srobovanie.STAV.M4_Moment_ToleranciaMAX.8:= P1_Srobovanie.PAR.M4_AtlasCopcoInputs[3].16;
//    P1_Srobovanie.STAV.M4_Moment_ToleranciaMAX.9:= P1_Srobovanie.PAR.M4_AtlasCopcoInputs[3].17;
//    P1_Srobovanie.STAV.M4_Moment_ToleranciaMAX.10:= P1_Srobovanie.PAR.M4_AtlasCopcoInputs[3].18;
//    P1_Srobovanie.STAV.M4_Moment_ToleranciaMAX.11:= P1_Srobovanie.PAR.M4_AtlasCopcoInputs[3].19;
//    P1_Srobovanie.STAV.M4_Moment_ToleranciaMAX.12:= P1_Srobovanie.PAR.M4_AtlasCopcoInputs[3].20;
//    P1_Srobovanie.STAV.M4_Moment_ToleranciaMAX.13:= P1_Srobovanie.PAR.M4_AtlasCopcoInputs[3].21;
//    P1_Srobovanie.STAV.M4_Moment_ToleranciaMAX.14:= P1_Srobovanie.PAR.M4_AtlasCopcoInputs[3].22;
//    P1_Srobovanie.STAV.M4_Moment_ToleranciaMAX.15:= P1_Srobovanie.PAR.M4_AtlasCopcoInputs[3].23;
//    P1_Srobovanie.STAV.M4_Moment_ToleranciaMAX.16:= P1_Srobovanie.PAR.M4_AtlasCopcoInputs[3].8;
//    P1_Srobovanie.STAV.M4_Moment_ToleranciaMAX.17:= P1_Srobovanie.PAR.M4_AtlasCopcoInputs[3].9;
//    P1_Srobovanie.STAV.M4_Moment_ToleranciaMAX.18:= P1_Srobovanie.PAR.M4_AtlasCopcoInputs[3].10;
//    P1_Srobovanie.STAV.M4_Moment_ToleranciaMAX.19:= P1_Srobovanie.PAR.M4_AtlasCopcoInputs[3].11;
//    P1_Srobovanie.STAV.M4_Moment_ToleranciaMAX.20:= P1_Srobovanie.PAR.M4_AtlasCopcoInputs[3].12;
//    P1_Srobovanie.STAV.M4_Moment_ToleranciaMAX.21:= P1_Srobovanie.PAR.M4_AtlasCopcoInputs[3].13;
//    P1_Srobovanie.STAV.M4_Moment_ToleranciaMAX.22:= P1_Srobovanie.PAR.M4_AtlasCopcoInputs[3].14;
//    P1_Srobovanie.STAV.M4_Moment_ToleranciaMAX.23:= P1_Srobovanie.PAR.M4_AtlasCopcoInputs[3].15;
//    P1_Srobovanie.STAV.M4_Moment_ToleranciaMAX.24:= P1_Srobovanie.PAR.M4_AtlasCopcoInputs[3].0;
//    P1_Srobovanie.STAV.M4_Moment_ToleranciaMAX.25:= P1_Srobovanie.PAR.M4_AtlasCopcoInputs[3].1;
//    P1_Srobovanie.STAV.M4_Moment_ToleranciaMAX.26:= P1_Srobovanie.PAR.M4_AtlasCopcoInputs[3].2;
//    P1_Srobovanie.STAV.M4_Moment_ToleranciaMAX.27:= P1_Srobovanie.PAR.M4_AtlasCopcoInputs[3].3;
//    P1_Srobovanie.STAV.M4_Moment_ToleranciaMAX.28:= P1_Srobovanie.PAR.M4_AtlasCopcoInputs[3].4;
//    P1_Srobovanie.STAV.M4_Moment_ToleranciaMAX.29:= P1_Srobovanie.PAR.M4_AtlasCopcoInputs[3].5;
//    P1_Srobovanie.STAV.M4_Moment_ToleranciaMAX.30:= P1_Srobovanie.PAR.M4_AtlasCopcoInputs[3].6;
//    P1_Srobovanie.STAV.M4_Moment_ToleranciaMAX.31:= P1_Srobovanie.PAR.M4_AtlasCopcoInputs[3].7;
//    M4_Moment_ToleranciaMAX_REAL:= UDINT_TO_REAL(P1_Srobovanie.STAV.M4_Moment_ToleranciaMAX);
//    IF M4_Moment_ToleranciaMAX_REAL > 0 THEN
//        P1_Srobovanie.STAV.M4_Moment_ToleranciaMAX_REAL:= (M4_Moment_ToleranciaMAX_REAL*0.65)/42598;
//    ELSE
//        P1_Srobovanie.STAV.M4_Moment_ToleranciaMAX_REAL:= 0.0;
//    END_IF
    (*P1_Srobovanie.STAV.M4_Moment_ToleranciaMAX_REAL:= M4_Moment_ToleranciaMAX_REAL/100;*)

    M4_PrevodMomentu.AtlasMaximalnaTolerancia:=P1_Srobovanie.PAR.M4_AtlasCopcoInputs[3];
    P1_Srobovanie.STAV.M4_Moment_ToleranciaMAX_REAL:=M4_PrevodMomentu.ToleranciaMAX;

    //Moment - Tolerancia MIN//
//    P1_Srobovanie.STAV.M4_Moment_ToleranciaMIN.0:= P1_Srobovanie.PAR.M4_AtlasCopcoInputs[4].24;
//    P1_Srobovanie.STAV.M4_Moment_ToleranciaMIN.1:= P1_Srobovanie.PAR.M4_AtlasCopcoInputs[4].25;
//    P1_Srobovanie.STAV.M4_Moment_ToleranciaMIN.2:= P1_Srobovanie.PAR.M4_AtlasCopcoInputs[4].26;
//    P1_Srobovanie.STAV.M4_Moment_ToleranciaMIN.3:= P1_Srobovanie.PAR.M4_AtlasCopcoInputs[4].27;
//    P1_Srobovanie.STAV.M4_Moment_ToleranciaMIN.4:= P1_Srobovanie.PAR.M4_AtlasCopcoInputs[4].28;
//    P1_Srobovanie.STAV.M4_Moment_ToleranciaMIN.5:= P1_Srobovanie.PAR.M4_AtlasCopcoInputs[4].29;
//    P1_Srobovanie.STAV.M4_Moment_ToleranciaMIN.6:= P1_Srobovanie.PAR.M4_AtlasCopcoInputs[4].30;
//    P1_Srobovanie.STAV.M4_Moment_ToleranciaMIN.7:= P1_Srobovanie.PAR.M4_AtlasCopcoInputs[4].31;
//    P1_Srobovanie.STAV.M4_Moment_ToleranciaMIN.8:= P1_Srobovanie.PAR.M4_AtlasCopcoInputs[4].16;
//    P1_Srobovanie.STAV.M4_Moment_ToleranciaMIN.9:= P1_Srobovanie.PAR.M4_AtlasCopcoInputs[4].17;
//    P1_Srobovanie.STAV.M4_Moment_ToleranciaMIN.10:= P1_Srobovanie.PAR.M4_AtlasCopcoInputs[4].18;
//    P1_Srobovanie.STAV.M4_Moment_ToleranciaMIN.11:= P1_Srobovanie.PAR.M4_AtlasCopcoInputs[4].19;
//    P1_Srobovanie.STAV.M4_Moment_ToleranciaMIN.12:= P1_Srobovanie.PAR.M4_AtlasCopcoInputs[4].20;
//    P1_Srobovanie.STAV.M4_Moment_ToleranciaMIN.13:= P1_Srobovanie.PAR.M4_AtlasCopcoInputs[4].21;
//    P1_Srobovanie.STAV.M4_Moment_ToleranciaMIN.14:= P1_Srobovanie.PAR.M4_AtlasCopcoInputs[4].22;
//    P1_Srobovanie.STAV.M4_Moment_ToleranciaMIN.15:= P1_Srobovanie.PAR.M4_AtlasCopcoInputs[4].23;
//    P1_Srobovanie.STAV.M4_Moment_ToleranciaMIN.16:= P1_Srobovanie.PAR.M4_AtlasCopcoInputs[4].8;
//    P1_Srobovanie.STAV.M4_Moment_ToleranciaMIN.17:= P1_Srobovanie.PAR.M4_AtlasCopcoInputs[4].9;
//    P1_Srobovanie.STAV.M4_Moment_ToleranciaMIN.18:= P1_Srobovanie.PAR.M4_AtlasCopcoInputs[4].10;
//    P1_Srobovanie.STAV.M4_Moment_ToleranciaMIN.19:= P1_Srobovanie.PAR.M4_AtlasCopcoInputs[4].11;
//    P1_Srobovanie.STAV.M4_Moment_ToleranciaMIN.20:= P1_Srobovanie.PAR.M4_AtlasCopcoInputs[4].12;
//    P1_Srobovanie.STAV.M4_Moment_ToleranciaMIN.21:= P1_Srobovanie.PAR.M4_AtlasCopcoInputs[4].13;
//    P1_Srobovanie.STAV.M4_Moment_ToleranciaMIN.22:= P1_Srobovanie.PAR.M4_AtlasCopcoInputs[4].14;
//    P1_Srobovanie.STAV.M4_Moment_ToleranciaMIN.23:= P1_Srobovanie.PAR.M4_AtlasCopcoInputs[4].15;
//    P1_Srobovanie.STAV.M4_Moment_ToleranciaMIN.24:= P1_Srobovanie.PAR.M4_AtlasCopcoInputs[4].0;
//    P1_Srobovanie.STAV.M4_Moment_ToleranciaMIN.25:= P1_Srobovanie.PAR.M4_AtlasCopcoInputs[4].1;
//    P1_Srobovanie.STAV.M4_Moment_ToleranciaMIN.26:= P1_Srobovanie.PAR.M4_AtlasCopcoInputs[4].2;
//    P1_Srobovanie.STAV.M4_Moment_ToleranciaMIN.27:= P1_Srobovanie.PAR.M4_AtlasCopcoInputs[4].3;
//    P1_Srobovanie.STAV.M4_Moment_ToleranciaMIN.28:= P1_Srobovanie.PAR.M4_AtlasCopcoInputs[4].4;
//    P1_Srobovanie.STAV.M4_Moment_ToleranciaMIN.29:= P1_Srobovanie.PAR.M4_AtlasCopcoInputs[4].5;
//    P1_Srobovanie.STAV.M4_Moment_ToleranciaMIN.30:= P1_Srobovanie.PAR.M4_AtlasCopcoInputs[4].6;
//    P1_Srobovanie.STAV.M4_Moment_ToleranciaMIN.31:= P1_Srobovanie.PAR.M4_AtlasCopcoInputs[4].7;
//    M4_Moment_ToleranciaMIN_REAL:= UDINT_TO_REAL(P1_Srobovanie.STAV.M4_Moment_ToleranciaMIN);
//    IF M4_Moment_ToleranciaMIN_REAL > 0 THEN
//        P1_Srobovanie.STAV.M4_Moment_ToleranciaMIN_REAL:= (M4_Moment_ToleranciaMIN_REAL*0.65)/42598;
//    ELSE
//        P1_Srobovanie.STAV.M4_Moment_ToleranciaMIN_REAL:= 0.0;
//    END_IF
//
//
    (*P1_Srobovanie.STAV.M4_Moment_ToleranciaMIN_REAL:= M4_Moment_ToleranciaMIN_REAL /100;*)

    M4_PrevodMomentu.AtlasMinimalnaTolerancia:=P1_Srobovanie.PAR.M4_AtlasCopcoInputs[4];
    P1_Srobovanie.STAV.M4_Moment_ToleranciaMIN_REAL:=M4_PrevodMomentu.ToleranciaMIN;

    //Dosiahnutý úhol//
    P1_Srobovanie.STAV.M4_DosiahnutyUhol.0:= P1_Srobovanie.PAR.M4_AtlasCopcoInputs[0].24;
    P1_Srobovanie.STAV.M4_DosiahnutyUhol.1:= P1_Srobovanie.PAR.M4_AtlasCopcoInputs[0].25;
    P1_Srobovanie.STAV.M4_DosiahnutyUhol.2:= P1_Srobovanie.PAR.M4_AtlasCopcoInputs[0].26;
    P1_Srobovanie.STAV.M4_DosiahnutyUhol.3:= P1_Srobovanie.PAR.M4_AtlasCopcoInputs[0].27;
    P1_Srobovanie.STAV.M4_DosiahnutyUhol.4:= P1_Srobovanie.PAR.M4_AtlasCopcoInputs[0].28;
    P1_Srobovanie.STAV.M4_DosiahnutyUhol.5:= P1_Srobovanie.PAR.M4_AtlasCopcoInputs[0].29;
    P1_Srobovanie.STAV.M4_DosiahnutyUhol.6:= P1_Srobovanie.PAR.M4_AtlasCopcoInputs[0].30;
    P1_Srobovanie.STAV.M4_DosiahnutyUhol.7:= P1_Srobovanie.PAR.M4_AtlasCopcoInputs[0].31;
    P1_Srobovanie.STAV.M4_DosiahnutyUhol.8:= P1_Srobovanie.PAR.M4_AtlasCopcoInputs[0].16;
    P1_Srobovanie.STAV.M4_DosiahnutyUhol.9:= P1_Srobovanie.PAR.M4_AtlasCopcoInputs[0].17;
    P1_Srobovanie.STAV.M4_DosiahnutyUhol.10:= P1_Srobovanie.PAR.M4_AtlasCopcoInputs[0].18;
    P1_Srobovanie.STAV.M4_DosiahnutyUhol.11:= P1_Srobovanie.PAR.M4_AtlasCopcoInputs[0].19;
    P1_Srobovanie.STAV.M4_DosiahnutyUhol.12:= P1_Srobovanie.PAR.M4_AtlasCopcoInputs[0].20;
    P1_Srobovanie.STAV.M4_DosiahnutyUhol.13:= P1_Srobovanie.PAR.M4_AtlasCopcoInputs[0].21;
    P1_Srobovanie.STAV.M4_DosiahnutyUhol.14:= P1_Srobovanie.PAR.M4_AtlasCopcoInputs[0].22;
    P1_Srobovanie.STAV.M4_DosiahnutyUhol.15:= P1_Srobovanie.PAR.M4_AtlasCopcoInputs[0].23;

    //Uhol - Tolerancia MAX//
    P1_Srobovanie.STAV.M4_Uhol_ToleranciaMAX.0:= P1_Srobovanie.PAR.M4_AtlasCopcoInputs[2].8;
    P1_Srobovanie.STAV.M4_Uhol_ToleranciaMAX.1:= P1_Srobovanie.PAR.M4_AtlasCopcoInputs[2].9;
    P1_Srobovanie.STAV.M4_Uhol_ToleranciaMAX.2:= P1_Srobovanie.PAR.M4_AtlasCopcoInputs[2].10;
    P1_Srobovanie.STAV.M4_Uhol_ToleranciaMAX.3:= P1_Srobovanie.PAR.M4_AtlasCopcoInputs[2].11;
    P1_Srobovanie.STAV.M4_Uhol_ToleranciaMAX.4:= P1_Srobovanie.PAR.M4_AtlasCopcoInputs[2].12;
    P1_Srobovanie.STAV.M4_Uhol_ToleranciaMAX.5:= P1_Srobovanie.PAR.M4_AtlasCopcoInputs[2].13;
    P1_Srobovanie.STAV.M4_Uhol_ToleranciaMAX.6:= P1_Srobovanie.PAR.M4_AtlasCopcoInputs[2].14;
    P1_Srobovanie.STAV.M4_Uhol_ToleranciaMAX.7:= P1_Srobovanie.PAR.M4_AtlasCopcoInputs[2].15;
    P1_Srobovanie.STAV.M4_Uhol_ToleranciaMAX.8:= P1_Srobovanie.PAR.M4_AtlasCopcoInputs[2].0;
    P1_Srobovanie.STAV.M4_Uhol_ToleranciaMAX.9:= P1_Srobovanie.PAR.M4_AtlasCopcoInputs[2].1;
    P1_Srobovanie.STAV.M4_Uhol_ToleranciaMAX.10:= P1_Srobovanie.PAR.M4_AtlasCopcoInputs[2].2;
    P1_Srobovanie.STAV.M4_Uhol_ToleranciaMAX.11:= P1_Srobovanie.PAR.M4_AtlasCopcoInputs[2].3;
    P1_Srobovanie.STAV.M4_Uhol_ToleranciaMAX.12:= P1_Srobovanie.PAR.M4_AtlasCopcoInputs[2].4;
    P1_Srobovanie.STAV.M4_Uhol_ToleranciaMAX.13:= P1_Srobovanie.PAR.M4_AtlasCopcoInputs[2].5;
    P1_Srobovanie.STAV.M4_Uhol_ToleranciaMAX.14:= P1_Srobovanie.PAR.M4_AtlasCopcoInputs[2].6;
    P1_Srobovanie.STAV.M4_Uhol_ToleranciaMAX.15:= P1_Srobovanie.PAR.M4_AtlasCopcoInputs[2].7;

    //Uhol - Tolerancia MIN//
    P1_Srobovanie.STAV.M4_Uhol_ToleranciaMIN.0:= P1_Srobovanie.PAR.M4_AtlasCopcoInputs[2].24;
    P1_Srobovanie.STAV.M4_Uhol_ToleranciaMIN.1:= P1_Srobovanie.PAR.M4_AtlasCopcoInputs[2].25;
    P1_Srobovanie.STAV.M4_Uhol_ToleranciaMIN.2:= P1_Srobovanie.PAR.M4_AtlasCopcoInputs[2].26;
    P1_Srobovanie.STAV.M4_Uhol_ToleranciaMIN.3:= P1_Srobovanie.PAR.M4_AtlasCopcoInputs[2].27;
    P1_Srobovanie.STAV.M4_Uhol_ToleranciaMIN.4:= P1_Srobovanie.PAR.M4_AtlasCopcoInputs[2].28;
    P1_Srobovanie.STAV.M4_Uhol_ToleranciaMIN.5:= P1_Srobovanie.PAR.M4_AtlasCopcoInputs[2].29;
    P1_Srobovanie.STAV.M4_Uhol_ToleranciaMIN.6:= P1_Srobovanie.PAR.M4_AtlasCopcoInputs[2].30;
    P1_Srobovanie.STAV.M4_Uhol_ToleranciaMIN.7:= P1_Srobovanie.PAR.M4_AtlasCopcoInputs[2].31;
    P1_Srobovanie.STAV.M4_Uhol_ToleranciaMIN.8:= P1_Srobovanie.PAR.M4_AtlasCopcoInputs[2].16;
    P1_Srobovanie.STAV.M4_Uhol_ToleranciaMIN.9:= P1_Srobovanie.PAR.M4_AtlasCopcoInputs[2].17;
    P1_Srobovanie.STAV.M4_Uhol_ToleranciaMIN.10:= P1_Srobovanie.PAR.M4_AtlasCopcoInputs[2].18;
    P1_Srobovanie.STAV.M4_Uhol_ToleranciaMIN.11:= P1_Srobovanie.PAR.M4_AtlasCopcoInputs[2].19;
    P1_Srobovanie.STAV.M4_Uhol_ToleranciaMIN.12:= P1_Srobovanie.PAR.M4_AtlasCopcoInputs[2].20;
    P1_Srobovanie.STAV.M4_Uhol_ToleranciaMIN.13:= P1_Srobovanie.PAR.M4_AtlasCopcoInputs[2].21;
    P1_Srobovanie.STAV.M4_Uhol_ToleranciaMIN.14:= P1_Srobovanie.PAR.M4_AtlasCopcoInputs[2].22;
    P1_Srobovanie.STAV.M4_Uhol_ToleranciaMIN.15:= P1_Srobovanie.PAR.M4_AtlasCopcoInputs[2].23;

    //*********************************Skrutkovacka K30*******************************************************************************//
    //Vstupy z AtlasCopco do PLC//
    P1_Srobovanie.Skrutkovacka_K30.Stav_VysledokPotvrdeny:= P1_Srobovanie.PAR.K30_AtlasCopcoInputs[0].0;
    P1_Srobovanie.Skrutkovacka_K30.Stav_EmergencyStop:= P1_Srobovanie.PAR.K30_AtlasCopcoInputs[0].1;
    P1_Srobovanie.Skrutkovacka_K30.Stav_READY_to_START:= P1_Srobovanie.PAR.K30_AtlasCopcoInputs[0].2;
    P1_Srobovanie.Skrutkovacka_K30.Stav_MANUAL:= P1_Srobovanie.PAR.K30_AtlasCopcoInputs[0].3;
    P1_Srobovanie.Skrutkovacka_K30.Stav_UtahovanieUkoncene:= P1_Srobovanie.PAR.K30_AtlasCopcoInputs[0].4;
    P1_Srobovanie.Skrutkovacka_K30.Stav_VysledokUtahovania_NG:= P1_Srobovanie.PAR.K30_AtlasCopcoInputs[0].5;
    P1_Srobovanie.Skrutkovacka_K30.Stav_VysledokUtahovania_OK:= P1_Srobovanie.PAR.K30_AtlasCopcoInputs[0].6;
    P1_Srobovanie.Skrutkovacka_K30.Stav_SmerOtacania_VPRED:= P1_Srobovanie.PAR.K30_AtlasCopcoInputs[0].7;
    P1_Srobovanie.Skrutkovacka_K30.Stav_BUSY:= P1_Srobovanie.PAR.K30_AtlasCopcoInputs[0].8; //Další byte
    P1_Srobovanie.Skrutkovacka_K30.Stav_ControlerSwitch_ON:= P1_Srobovanie.PAR.K30_AtlasCopcoInputs[0].9;
    P1_Srobovanie.Skrutkovacka_K30.Stav_Station_READY:= P1_Srobovanie.PAR.K30_AtlasCopcoInputs[0].10;
    P1_Srobovanie.Skrutkovacka_K30.Stav_NastrojPripojeny:= P1_Srobovanie.PAR.K30_AtlasCopcoInputs[0].11;
    P1_Srobovanie.Skrutkovacka_K30.Stav_NastrojUtahuje:= P1_Srobovanie.PAR.K30_AtlasCopcoInputs[0].12;

    //Výstupy z PLC do AtlasCopco//
    P1_Srobovanie.PAR.K30_AtlasCopcoOutputs[0].0:= P1_Srobovanie.Skrutkovacka_K30.RESET_Poruchy;
    P1_Srobovanie.PAR.K30_AtlasCopcoOutputs[0].1:= P1_Srobovanie.Skrutkovacka_K30.RESET_Vysledkov;
    P1_Srobovanie.PAR.K30_AtlasCopcoOutputs[0].2:= P1_Srobovanie.Skrutkovacka_K30.START_Skrutkovania;
    P1_Srobovanie.PAR.K30_AtlasCopcoOutputs[0].3:= P1_Srobovanie.Skrutkovacka_K30.START_Utahovania;

    //Dosiahnutý moment//
//    P1_Srobovanie.STAV.K30_DosiahnutyMoment.0:= P1_Srobovanie.PAR.K30_AtlasCopcoInputs[1].24;
//    P1_Srobovanie.STAV.K30_DosiahnutyMoment.1:= P1_Srobovanie.PAR.K30_AtlasCopcoInputs[1].25;
//    P1_Srobovanie.STAV.K30_DosiahnutyMoment.2:= P1_Srobovanie.PAR.K30_AtlasCopcoInputs[1].26;
//    P1_Srobovanie.STAV.K30_DosiahnutyMoment.3:= P1_Srobovanie.PAR.K30_AtlasCopcoInputs[1].27;
//    P1_Srobovanie.STAV.K30_DosiahnutyMoment.4:= P1_Srobovanie.PAR.K30_AtlasCopcoInputs[1].28;
//    P1_Srobovanie.STAV.K30_DosiahnutyMoment.5:= P1_Srobovanie.PAR.K30_AtlasCopcoInputs[1].29;
//    P1_Srobovanie.STAV.K30_DosiahnutyMoment.6:= P1_Srobovanie.PAR.K30_AtlasCopcoInputs[1].30;
//    P1_Srobovanie.STAV.K30_DosiahnutyMoment.7:= P1_Srobovanie.PAR.K30_AtlasCopcoInputs[1].31;
//    P1_Srobovanie.STAV.K30_DosiahnutyMoment.8:= P1_Srobovanie.PAR.K30_AtlasCopcoInputs[1].16;
//    P1_Srobovanie.STAV.K30_DosiahnutyMoment.9:= P1_Srobovanie.PAR.K30_AtlasCopcoInputs[1].17;
//    P1_Srobovanie.STAV.K30_DosiahnutyMoment.10:= P1_Srobovanie.PAR.K30_AtlasCopcoInputs[1].18;
//    P1_Srobovanie.STAV.K30_DosiahnutyMoment.11:= P1_Srobovanie.PAR.K30_AtlasCopcoInputs[1].19;
//    P1_Srobovanie.STAV.K30_DosiahnutyMoment.12:= P1_Srobovanie.PAR.K30_AtlasCopcoInputs[1].20;
//    P1_Srobovanie.STAV.K30_DosiahnutyMoment.13:= P1_Srobovanie.PAR.K30_AtlasCopcoInputs[1].21;
//    P1_Srobovanie.STAV.K30_DosiahnutyMoment.14:= P1_Srobovanie.PAR.K30_AtlasCopcoInputs[1].22;
//    P1_Srobovanie.STAV.K30_DosiahnutyMoment.15:= P1_Srobovanie.PAR.K30_AtlasCopcoInputs[1].23;
//    P1_Srobovanie.STAV.K30_DosiahnutyMoment.16:= P1_Srobovanie.PAR.K30_AtlasCopcoInputs[1].8;
//    P1_Srobovanie.STAV.K30_DosiahnutyMoment.17:= P1_Srobovanie.PAR.K30_AtlasCopcoInputs[1].9;
//    P1_Srobovanie.STAV.K30_DosiahnutyMoment.18:= P1_Srobovanie.PAR.K30_AtlasCopcoInputs[1].10;
//    P1_Srobovanie.STAV.K30_DosiahnutyMoment.19:= P1_Srobovanie.PAR.K30_AtlasCopcoInputs[1].11;
//    P1_Srobovanie.STAV.K30_DosiahnutyMoment.20:= P1_Srobovanie.PAR.K30_AtlasCopcoInputs[1].12;
//    P1_Srobovanie.STAV.K30_DosiahnutyMoment.21:= P1_Srobovanie.PAR.K30_AtlasCopcoInputs[1].13;
//    P1_Srobovanie.STAV.K30_DosiahnutyMoment.22:= P1_Srobovanie.PAR.K30_AtlasCopcoInputs[1].14;
//    P1_Srobovanie.STAV.K30_DosiahnutyMoment.23:= P1_Srobovanie.PAR.K30_AtlasCopcoInputs[1].15;
//    P1_Srobovanie.STAV.K30_DosiahnutyMoment.24:= P1_Srobovanie.PAR.K30_AtlasCopcoInputs[1].0;
//    P1_Srobovanie.STAV.K30_DosiahnutyMoment.25:= P1_Srobovanie.PAR.K30_AtlasCopcoInputs[1].1;
//    P1_Srobovanie.STAV.K30_DosiahnutyMoment.26:= P1_Srobovanie.PAR.K30_AtlasCopcoInputs[1].2;
//    P1_Srobovanie.STAV.K30_DosiahnutyMoment.27:= P1_Srobovanie.PAR.K30_AtlasCopcoInputs[1].3;
//    P1_Srobovanie.STAV.K30_DosiahnutyMoment.28:= P1_Srobovanie.PAR.K30_AtlasCopcoInputs[1].4;
//    P1_Srobovanie.STAV.K30_DosiahnutyMoment.29:= P1_Srobovanie.PAR.K30_AtlasCopcoInputs[1].5;
//    P1_Srobovanie.STAV.K30_DosiahnutyMoment.30:= P1_Srobovanie.PAR.K30_AtlasCopcoInputs[1].6;
//    P1_Srobovanie.STAV.K30_DosiahnutyMoment.31:= P1_Srobovanie.PAR.K30_AtlasCopcoInputs[1].7;
//    K30_DosiahnutyMoment_REAL:= UDINT_TO_REAL(P1_Srobovanie.STAV.K30_DosiahnutyMoment);
//    IF K30_DosiahnutyMoment_REAL > 0 THEN
//        P1_Srobovanie.STAV.K30_DosiahnutyMoment_REAL:= K30_DosiahnutyMoment_REAL/100;
//    ELSE
//        P1_Srobovanie.STAV.K30_DosiahnutyMoment_REAL:= 0.0;
//    END_IF

    (*P1_Srobovanie.STAV.K30_DosiahnutyMoment_REAL:= (K30_DosiahnutyMoment_REAL*0.65)/42598;*)

    K30_PrevodMomentu.AtlasAktualnyMoment:=P1_Srobovanie.PAR.K30_AtlasCopcoInputs[1];
    P1_Srobovanie.STAV.K30_DosiahnutyMoment_REAL:=K30_PrevodMomentu.AktualnyMoment;

    //Moment - Tolerancia MAX//
//    P1_Srobovanie.STAV.K30_Moment_ToleranciaMAX.0:= P1_Srobovanie.PAR.K30_AtlasCopcoInputs[3].24;
//    P1_Srobovanie.STAV.K30_Moment_ToleranciaMAX.1:= P1_Srobovanie.PAR.K30_AtlasCopcoInputs[3].25;
//    P1_Srobovanie.STAV.K30_Moment_ToleranciaMAX.2:= P1_Srobovanie.PAR.K30_AtlasCopcoInputs[3].26;
//    P1_Srobovanie.STAV.K30_Moment_ToleranciaMAX.3:= P1_Srobovanie.PAR.K30_AtlasCopcoInputs[3].27;
//    P1_Srobovanie.STAV.K30_Moment_ToleranciaMAX.4:= P1_Srobovanie.PAR.K30_AtlasCopcoInputs[3].28;
//    P1_Srobovanie.STAV.K30_Moment_ToleranciaMAX.5:= P1_Srobovanie.PAR.K30_AtlasCopcoInputs[3].29;
//    P1_Srobovanie.STAV.K30_Moment_ToleranciaMAX.6:= P1_Srobovanie.PAR.K30_AtlasCopcoInputs[3].30;
//    P1_Srobovanie.STAV.K30_Moment_ToleranciaMAX.7:= P1_Srobovanie.PAR.K30_AtlasCopcoInputs[3].31;
//    P1_Srobovanie.STAV.K30_Moment_ToleranciaMAX.8:= P1_Srobovanie.PAR.K30_AtlasCopcoInputs[3].16;
//    P1_Srobovanie.STAV.K30_Moment_ToleranciaMAX.9:= P1_Srobovanie.PAR.K30_AtlasCopcoInputs[3].17;
//    P1_Srobovanie.STAV.K30_Moment_ToleranciaMAX.10:= P1_Srobovanie.PAR.K30_AtlasCopcoInputs[3].18;
//    P1_Srobovanie.STAV.K30_Moment_ToleranciaMAX.11:= P1_Srobovanie.PAR.K30_AtlasCopcoInputs[3].19;
//    P1_Srobovanie.STAV.K30_Moment_ToleranciaMAX.12:= P1_Srobovanie.PAR.K30_AtlasCopcoInputs[3].20;
//    P1_Srobovanie.STAV.K30_Moment_ToleranciaMAX.13:= P1_Srobovanie.PAR.K30_AtlasCopcoInputs[3].21;
//    P1_Srobovanie.STAV.K30_Moment_ToleranciaMAX.14:= P1_Srobovanie.PAR.K30_AtlasCopcoInputs[3].22;
//    P1_Srobovanie.STAV.K30_Moment_ToleranciaMAX.15:= P1_Srobovanie.PAR.K30_AtlasCopcoInputs[3].23;
//    P1_Srobovanie.STAV.K30_Moment_ToleranciaMAX.16:= P1_Srobovanie.PAR.K30_AtlasCopcoInputs[3].8;
//    P1_Srobovanie.STAV.K30_Moment_ToleranciaMAX.17:= P1_Srobovanie.PAR.K30_AtlasCopcoInputs[3].9;
//    P1_Srobovanie.STAV.K30_Moment_ToleranciaMAX.18:= P1_Srobovanie.PAR.K30_AtlasCopcoInputs[3].10;
//    P1_Srobovanie.STAV.K30_Moment_ToleranciaMAX.19:= P1_Srobovanie.PAR.K30_AtlasCopcoInputs[3].11;
//    P1_Srobovanie.STAV.K30_Moment_ToleranciaMAX.20:= P1_Srobovanie.PAR.K30_AtlasCopcoInputs[3].12;
//    P1_Srobovanie.STAV.K30_Moment_ToleranciaMAX.21:= P1_Srobovanie.PAR.K30_AtlasCopcoInputs[3].13;
//    P1_Srobovanie.STAV.K30_Moment_ToleranciaMAX.22:= P1_Srobovanie.PAR.K30_AtlasCopcoInputs[3].14;
//    P1_Srobovanie.STAV.K30_Moment_ToleranciaMAX.23:= P1_Srobovanie.PAR.K30_AtlasCopcoInputs[3].15;
//    P1_Srobovanie.STAV.K30_Moment_ToleranciaMAX.24:= P1_Srobovanie.PAR.K30_AtlasCopcoInputs[3].0;
//    P1_Srobovanie.STAV.K30_Moment_ToleranciaMAX.25:= P1_Srobovanie.PAR.K30_AtlasCopcoInputs[3].1;
//    P1_Srobovanie.STAV.K30_Moment_ToleranciaMAX.26:= P1_Srobovanie.PAR.K30_AtlasCopcoInputs[3].2;
//    P1_Srobovanie.STAV.K30_Moment_ToleranciaMAX.27:= P1_Srobovanie.PAR.K30_AtlasCopcoInputs[3].3;
//    P1_Srobovanie.STAV.K30_Moment_ToleranciaMAX.28:= P1_Srobovanie.PAR.K30_AtlasCopcoInputs[3].4;
//    P1_Srobovanie.STAV.K30_Moment_ToleranciaMAX.29:= P1_Srobovanie.PAR.K30_AtlasCopcoInputs[3].5;
//    P1_Srobovanie.STAV.K30_Moment_ToleranciaMAX.30:= P1_Srobovanie.PAR.K30_AtlasCopcoInputs[3].6;
//    P1_Srobovanie.STAV.K30_Moment_ToleranciaMAX.31:= P1_Srobovanie.PAR.K30_AtlasCopcoInputs[3].7;
//    K30_Moment_ToleranciaMAX_REAL:= UDINT_TO_REAL(P1_Srobovanie.STAV.K30_Moment_ToleranciaMAX);
//    IF K30_Moment_ToleranciaMAX_REAL > 0 THEN
//       P1_Srobovanie.STAV.K30_Moment_ToleranciaMAX_REAL:= K30_Moment_ToleranciaMAX_REAL/100;
//    ELSE
//        P1_Srobovanie.STAV.K30_Moment_ToleranciaMAX_REAL:= 0.0;
//    END_IF

    (*P1_Srobovanie.STAV.K30_Moment_ToleranciaMAX_REAL:= (K30_Moment_ToleranciaMAX_REAL*0.65)/42598;*)
    K30_PrevodMomentu.AtlasMaximalnaTolerancia:=P1_Srobovanie.PAR.K30_AtlasCopcoInputs[3];
    P1_Srobovanie.STAV.K30_Moment_ToleranciaMAX_REAL:=K30_PrevodMomentu.ToleranciaMAX;

    //Moment - Tolerancia MIN//
//    P1_Srobovanie.STAV.K30_Moment_ToleranciaMIN.0:= P1_Srobovanie.PAR.K30_AtlasCopcoInputs[4].24;
//    P1_Srobovanie.STAV.K30_Moment_ToleranciaMIN.1:= P1_Srobovanie.PAR.K30_AtlasCopcoInputs[4].25;
//    P1_Srobovanie.STAV.K30_Moment_ToleranciaMIN.2:= P1_Srobovanie.PAR.K30_AtlasCopcoInputs[4].26;
//    P1_Srobovanie.STAV.K30_Moment_ToleranciaMIN.3:= P1_Srobovanie.PAR.K30_AtlasCopcoInputs[4].27;
//    P1_Srobovanie.STAV.K30_Moment_ToleranciaMIN.4:= P1_Srobovanie.PAR.K30_AtlasCopcoInputs[4].28;
//    P1_Srobovanie.STAV.K30_Moment_ToleranciaMIN.5:= P1_Srobovanie.PAR.K30_AtlasCopcoInputs[4].29;
//    P1_Srobovanie.STAV.K30_Moment_ToleranciaMIN.6:= P1_Srobovanie.PAR.K30_AtlasCopcoInputs[4].30;
//    P1_Srobovanie.STAV.K30_Moment_ToleranciaMIN.7:= P1_Srobovanie.PAR.K30_AtlasCopcoInputs[4].31;
//    P1_Srobovanie.STAV.K30_Moment_ToleranciaMIN.8:= P1_Srobovanie.PAR.K30_AtlasCopcoInputs[4].16;
//    P1_Srobovanie.STAV.K30_Moment_ToleranciaMIN.9:= P1_Srobovanie.PAR.K30_AtlasCopcoInputs[4].17;
//    P1_Srobovanie.STAV.K30_Moment_ToleranciaMIN.10:= P1_Srobovanie.PAR.K30_AtlasCopcoInputs[4].18;
//    P1_Srobovanie.STAV.K30_Moment_ToleranciaMIN.11:= P1_Srobovanie.PAR.K30_AtlasCopcoInputs[4].19;
//    P1_Srobovanie.STAV.K30_Moment_ToleranciaMIN.12:= P1_Srobovanie.PAR.K30_AtlasCopcoInputs[4].20;
//    P1_Srobovanie.STAV.K30_Moment_ToleranciaMIN.13:= P1_Srobovanie.PAR.K30_AtlasCopcoInputs[4].21;
//    P1_Srobovanie.STAV.K30_Moment_ToleranciaMIN.14:= P1_Srobovanie.PAR.K30_AtlasCopcoInputs[4].22;
//    P1_Srobovanie.STAV.K30_Moment_ToleranciaMIN.15:= P1_Srobovanie.PAR.K30_AtlasCopcoInputs[4].23;
//    P1_Srobovanie.STAV.K30_Moment_ToleranciaMIN.16:= P1_Srobovanie.PAR.K30_AtlasCopcoInputs[4].8;
//    P1_Srobovanie.STAV.K30_Moment_ToleranciaMIN.17:= P1_Srobovanie.PAR.K30_AtlasCopcoInputs[4].9;
//    P1_Srobovanie.STAV.K30_Moment_ToleranciaMIN.18:= P1_Srobovanie.PAR.K30_AtlasCopcoInputs[4].10;
//    P1_Srobovanie.STAV.K30_Moment_ToleranciaMIN.19:= P1_Srobovanie.PAR.K30_AtlasCopcoInputs[4].11;
//    P1_Srobovanie.STAV.K30_Moment_ToleranciaMIN.20:= P1_Srobovanie.PAR.K30_AtlasCopcoInputs[4].12;
//    P1_Srobovanie.STAV.K30_Moment_ToleranciaMIN.21:= P1_Srobovanie.PAR.K30_AtlasCopcoInputs[4].13;
//    P1_Srobovanie.STAV.K30_Moment_ToleranciaMIN.22:= P1_Srobovanie.PAR.K30_AtlasCopcoInputs[4].14;
//    P1_Srobovanie.STAV.K30_Moment_ToleranciaMIN.23:= P1_Srobovanie.PAR.K30_AtlasCopcoInputs[4].15;
//    P1_Srobovanie.STAV.K30_Moment_ToleranciaMIN.24:= P1_Srobovanie.PAR.K30_AtlasCopcoInputs[4].0;
//    P1_Srobovanie.STAV.K30_Moment_ToleranciaMIN.25:= P1_Srobovanie.PAR.K30_AtlasCopcoInputs[4].1;
//    P1_Srobovanie.STAV.K30_Moment_ToleranciaMIN.26:= P1_Srobovanie.PAR.K30_AtlasCopcoInputs[4].2;
//    P1_Srobovanie.STAV.K30_Moment_ToleranciaMIN.27:= P1_Srobovanie.PAR.K30_AtlasCopcoInputs[4].3;
//    P1_Srobovanie.STAV.K30_Moment_ToleranciaMIN.28:= P1_Srobovanie.PAR.K30_AtlasCopcoInputs[4].4;
//    P1_Srobovanie.STAV.K30_Moment_ToleranciaMIN.29:= P1_Srobovanie.PAR.K30_AtlasCopcoInputs[4].5;
//    P1_Srobovanie.STAV.K30_Moment_ToleranciaMIN.30:= P1_Srobovanie.PAR.K30_AtlasCopcoInputs[4].6;
//    P1_Srobovanie.STAV.K30_Moment_ToleranciaMIN.31:= P1_Srobovanie.PAR.K30_AtlasCopcoInputs[4].7;
//    K30_Moment_ToleranciaMIN_REAL:= UDINT_TO_REAL(P1_Srobovanie.STAV.K30_Moment_ToleranciaMIN);
//    IF K30_Moment_ToleranciaMIN_REAL > 0 THEN
//        P1_Srobovanie.STAV.K30_Moment_ToleranciaMIN_REAL:= K30_Moment_ToleranciaMIN_REAL /100;
//    ELSE
//        P1_Srobovanie.STAV.K30_Moment_ToleranciaMIN_REAL:= 0.0;
//    END_IF

    (*P1_Srobovanie.STAV.K30_Moment_ToleranciaMIN_REAL:= (K30_Moment_ToleranciaMIN_REAL*0.65)/42598;*)
    K30_PrevodMomentu.AtlasMinimalnaTolerancia:=P1_Srobovanie.PAR.K30_AtlasCopcoInputs[4];
    P1_Srobovanie.STAV.K30_Moment_ToleranciaMIN_REAL:=K30_PrevodMomentu.ToleranciaMIN;

    //Dosiahnutý úhol//
    P1_Srobovanie.STAV.K30_DosiahnutyUhol.0:= P1_Srobovanie.PAR.K30_AtlasCopcoInputs[0].24;
    P1_Srobovanie.STAV.K30_DosiahnutyUhol.1:= P1_Srobovanie.PAR.K30_AtlasCopcoInputs[0].25;
    P1_Srobovanie.STAV.K30_DosiahnutyUhol.2:= P1_Srobovanie.PAR.K30_AtlasCopcoInputs[0].26;
    P1_Srobovanie.STAV.K30_DosiahnutyUhol.3:= P1_Srobovanie.PAR.K30_AtlasCopcoInputs[0].27;
    P1_Srobovanie.STAV.K30_DosiahnutyUhol.4:= P1_Srobovanie.PAR.K30_AtlasCopcoInputs[0].28;
    P1_Srobovanie.STAV.K30_DosiahnutyUhol.5:= P1_Srobovanie.PAR.K30_AtlasCopcoInputs[0].29;
    P1_Srobovanie.STAV.K30_DosiahnutyUhol.6:= P1_Srobovanie.PAR.K30_AtlasCopcoInputs[0].30;
    P1_Srobovanie.STAV.K30_DosiahnutyUhol.7:= P1_Srobovanie.PAR.K30_AtlasCopcoInputs[0].31;
    P1_Srobovanie.STAV.K30_DosiahnutyUhol.8:= P1_Srobovanie.PAR.K30_AtlasCopcoInputs[0].16;
    P1_Srobovanie.STAV.K30_DosiahnutyUhol.9:= P1_Srobovanie.PAR.K30_AtlasCopcoInputs[0].17;
    P1_Srobovanie.STAV.K30_DosiahnutyUhol.10:= P1_Srobovanie.PAR.K30_AtlasCopcoInputs[0].18;
    P1_Srobovanie.STAV.K30_DosiahnutyUhol.11:= P1_Srobovanie.PAR.K30_AtlasCopcoInputs[0].19;
    P1_Srobovanie.STAV.K30_DosiahnutyUhol.12:= P1_Srobovanie.PAR.K30_AtlasCopcoInputs[0].20;
    P1_Srobovanie.STAV.K30_DosiahnutyUhol.13:= P1_Srobovanie.PAR.K30_AtlasCopcoInputs[0].21;
    P1_Srobovanie.STAV.K30_DosiahnutyUhol.14:= P1_Srobovanie.PAR.K30_AtlasCopcoInputs[0].22;
    P1_Srobovanie.STAV.K30_DosiahnutyUhol.15:= P1_Srobovanie.PAR.K30_AtlasCopcoInputs[0].23;

    //Uhol - Tolerancia MAX//
    P1_Srobovanie.STAV.K30_Uhol_ToleranciaMAX.0:= P1_Srobovanie.PAR.K30_AtlasCopcoInputs[2].8;
    P1_Srobovanie.STAV.K30_Uhol_ToleranciaMAX.1:= P1_Srobovanie.PAR.K30_AtlasCopcoInputs[2].9;
    P1_Srobovanie.STAV.K30_Uhol_ToleranciaMAX.2:= P1_Srobovanie.PAR.K30_AtlasCopcoInputs[2].10;
    P1_Srobovanie.STAV.K30_Uhol_ToleranciaMAX.3:= P1_Srobovanie.PAR.K30_AtlasCopcoInputs[2].11;
    P1_Srobovanie.STAV.K30_Uhol_ToleranciaMAX.4:= P1_Srobovanie.PAR.K30_AtlasCopcoInputs[2].12;
    P1_Srobovanie.STAV.K30_Uhol_ToleranciaMAX.5:= P1_Srobovanie.PAR.K30_AtlasCopcoInputs[2].13;
    P1_Srobovanie.STAV.K30_Uhol_ToleranciaMAX.6:= P1_Srobovanie.PAR.K30_AtlasCopcoInputs[2].14;
    P1_Srobovanie.STAV.K30_Uhol_ToleranciaMAX.7:= P1_Srobovanie.PAR.K30_AtlasCopcoInputs[2].15;
    P1_Srobovanie.STAV.K30_Uhol_ToleranciaMAX.8:= P1_Srobovanie.PAR.K30_AtlasCopcoInputs[2].0;
    P1_Srobovanie.STAV.K30_Uhol_ToleranciaMAX.9:= P1_Srobovanie.PAR.K30_AtlasCopcoInputs[2].1;
    P1_Srobovanie.STAV.K30_Uhol_ToleranciaMAX.10:= P1_Srobovanie.PAR.K30_AtlasCopcoInputs[2].2;
    P1_Srobovanie.STAV.K30_Uhol_ToleranciaMAX.11:= P1_Srobovanie.PAR.K30_AtlasCopcoInputs[2].3;
    P1_Srobovanie.STAV.K30_Uhol_ToleranciaMAX.12:= P1_Srobovanie.PAR.K30_AtlasCopcoInputs[2].4;
    P1_Srobovanie.STAV.K30_Uhol_ToleranciaMAX.13:= P1_Srobovanie.PAR.K30_AtlasCopcoInputs[2].5;
    P1_Srobovanie.STAV.K30_Uhol_ToleranciaMAX.14:= P1_Srobovanie.PAR.K30_AtlasCopcoInputs[2].6;
    P1_Srobovanie.STAV.K30_Uhol_ToleranciaMAX.15:= P1_Srobovanie.PAR.K30_AtlasCopcoInputs[2].7;

    //Uhol - Tolerancia MIN//
    P1_Srobovanie.STAV.K30_Uhol_ToleranciaMIN.0:= P1_Srobovanie.PAR.K30_AtlasCopcoInputs[2].24;
    P1_Srobovanie.STAV.K30_Uhol_ToleranciaMIN.1:= P1_Srobovanie.PAR.K30_AtlasCopcoInputs[2].25;
    P1_Srobovanie.STAV.K30_Uhol_ToleranciaMIN.2:= P1_Srobovanie.PAR.K30_AtlasCopcoInputs[2].26;
    P1_Srobovanie.STAV.K30_Uhol_ToleranciaMIN.3:= P1_Srobovanie.PAR.K30_AtlasCopcoInputs[2].27;
    P1_Srobovanie.STAV.K30_Uhol_ToleranciaMIN.4:= P1_Srobovanie.PAR.K30_AtlasCopcoInputs[2].28;
    P1_Srobovanie.STAV.K30_Uhol_ToleranciaMIN.5:= P1_Srobovanie.PAR.K30_AtlasCopcoInputs[2].29;
    P1_Srobovanie.STAV.K30_Uhol_ToleranciaMIN.6:= P1_Srobovanie.PAR.K30_AtlasCopcoInputs[2].30;
    P1_Srobovanie.STAV.K30_Uhol_ToleranciaMIN.7:= P1_Srobovanie.PAR.K30_AtlasCopcoInputs[2].31;
    P1_Srobovanie.STAV.K30_Uhol_ToleranciaMIN.8:= P1_Srobovanie.PAR.K30_AtlasCopcoInputs[2].16;
    P1_Srobovanie.STAV.K30_Uhol_ToleranciaMIN.9:= P1_Srobovanie.PAR.K30_AtlasCopcoInputs[2].17;
    P1_Srobovanie.STAV.K30_Uhol_ToleranciaMIN.10:= P1_Srobovanie.PAR.K30_AtlasCopcoInputs[2].18;
    P1_Srobovanie.STAV.K30_Uhol_ToleranciaMIN.11:= P1_Srobovanie.PAR.K30_AtlasCopcoInputs[2].19;
    P1_Srobovanie.STAV.K30_Uhol_ToleranciaMIN.12:= P1_Srobovanie.PAR.K30_AtlasCopcoInputs[2].20;
    P1_Srobovanie.STAV.K30_Uhol_ToleranciaMIN.13:= P1_Srobovanie.PAR.K30_AtlasCopcoInputs[2].21;
    P1_Srobovanie.STAV.K30_Uhol_ToleranciaMIN.14:= P1_Srobovanie.PAR.K30_AtlasCopcoInputs[2].22;
    P1_Srobovanie.STAV.K30_Uhol_ToleranciaMIN.15:= P1_Srobovanie.PAR.K30_AtlasCopcoInputs[2].23;

END_ACTION
```

#### OvlSkrutkovacichSetov.st
```iecst
ACTION OvlSkrutkovacichSetov:

	//***********************************Skrutkovací set K30************************************//
	//Volanie funkcie SequenceControl//
	SequenceControl(SC:= SC_SkrutkovaciSet_K30);

	CASE SC_SkrutkovaciSet_K30.Step OF

		0:
			SC_SkrutkovaciSet_K30.StepName:='0 - Nulovanie';
			P1_Srobovanie.SkrutSet_K30.Cmd.AutomatStart:= FALSE;
			P1_Srobovanie.SkrutSet_K30.Cmd.ManualStartHrniec:= FALSE;
			P1_Srobovanie.SkrutSet_K30.Cmd.PodajSkrutku:= FALSE;
			P1_Srobovanie.CMD.RR_SkrutSetK30_PodajSkrutku:= FALSE;
			P1_Srobovanie.CMD.RR_SkrutSetK30_Zasobnik_RUN:= FALSE;
			P1_Srobovanie.CMD.RR_SkrutSetK30_VysunBrzdu:= FALSE;
			P1_Srobovanie.SkrutSet_K30.Cmd.ManualPresunBrzdu:= FALSE;
			P1_Srobovanie.STAV.SkrutkaK30_READY:= FALSE;

			IF SC_P1_Srobovanie.Step <> 0 THEN
				SC_SkrutkovaciSet_K30.ResetStep:= TRUE;
				SC_SkrutkovaciSet_K30.Step:= 1;
			END_IF

		1:
			SC_SkrutkovaciSet_K30.StepName:='1 - Rozhodnutie o cinnosti';

			IF P1_Srobovanie.Automat THEN
				SC_SkrutkovaciSet_K30.ResetStep:= TRUE;
				SC_SkrutkovaciSet_K30.Step:= 10;
			ELSIF P1_Srobovanie.Manual THEN
				SC_SkrutkovaciSet_K30.ResetStep:= TRUE;
				SC_SkrutkovaciSet_K30.Step:= 20;
			END_IF

		10:
			SC_SkrutkovaciSet_K30.StepName:='10 - Automaticky rezim - cakam na signal podaj skrutku';
			SC_SkrutkovaciSet_K30.IdleTime.PT:= T#2s;
			SC_SkrutkovaciSet_K30.AlarmTime.PT:= T#5s;

			P1_Srobovanie.SkrutSet_K30.Cmd.AutomatStart:= TRUE;

			IF P1_Srobovanie.CMD.PodajSkrutku_K30 THEN
				P1_Srobovanie.CMD.PodajSkrutku_K30:= FALSE;
				SC_SkrutkovaciSet_K30.ResetStep:= TRUE;
				SC_SkrutkovaciSet_K30.Step:= 13;
			END_IF

		13:
			SC_SkrutkovaciSet_K30.StepName:='13 - Automaticky rezim - podanie skrutky do skrutkovacky';
			SC_SkrutkovaciSet_K30.IdleTime.PT:= T#2s;
			SC_SkrutkovaciSet_K30.AlarmTime.PT:= T#5s;

			IF NOT SC_SkrutkovaciSet_K30.Switch1 THEN
				P1_Srobovanie.SkrutSet_K30.Cmd.PodajSkrutku:= TRUE;
				SC_SkrutkovaciSet_K30.Switch1:= TRUE;
			END_IF

			IF P1_Srobovanie.SkrutSet_K30.Status.SkrutkaPripravena THEN
				P1_Srobovanie.STAV.SkrutkaK30_READY:= TRUE;
				P1_Srobovanie.SkrutSet_K30.Cmd.PodajSkrutku:= FALSE;
				SC_SkrutkovaciSet_K30.ResetStep:= TRUE;
				SC_SkrutkovaciSet_K30.Step:= 15;
			ELSIF P1_Srobovanie.SkrutSet_K30.Error.ErrorBit THEN
				P1_Srobovanie.SkrutSet_K30.Cmd.PodajSkrutku:= FALSE;
				P1_Alarmy[119]:= TRUE;
				P1_Pracovisko.STAV.Porucha_ST2:= TRUE;
			END_IF

		15:
			SC_SkrutkovaciSet_K30.StepName:='15 - Automaticky rezim - cakam na zrusenie stavu skrutka K30 READY';
			SC_SkrutkovaciSet_K30.IdleTime.PT:= T#2s;
			SC_SkrutkovaciSet_K30.AlarmTime.PT:= T#5s;

			IF NOT P1_Srobovanie.STAV.SkrutkaK30_READY THEN
				SC_SkrutkovaciSet_K30.ResetStep:= TRUE;
				SC_SkrutkovaciSet_K30.Step:= 10;
			ELSIF P1_Srobovanie.Manual THEN
				P1_Srobovanie.SkrutSet_K30.Cmd.AutomatStart:= FALSE;
				SC_SkrutkovaciSet_K30.ResetStep:= TRUE;
				SC_SkrutkovaciSet_K30.Step:= 20;
			END_IF

		20:
			SC_SkrutkovaciSet_K30.StepName:='20 - Manualny rezim';
			SC_SkrutkovaciSet_K30.IdleTime.PT:= T#2s;
			SC_SkrutkovaciSet_K30.AlarmTime.PT:= T#5s;

			//Ovládanie zásobníka//
			IF P1_Srobovanie.CMD.RR_SkrutSetK30_Zasobnik_RUN THEN
				P1_Srobovanie.SkrutSet_K30.Cmd.AutomatStart:= FALSE;
				P1_Srobovanie.SkrutSet_K30.Cmd.ManualStartHrniec:= TRUE;
			ELSE
				P1_Srobovanie.SkrutSet_K30.Cmd.ManualStartHrniec:= FALSE;
			END_IF

			//Ovládanie brzdy//
			IF P1_Srobovanie.CMD.RR_SkrutSetK30_VysunBrzdu THEN
				P1_Srobovanie.SkrutSet_K30.Cmd.AutomatStart:= FALSE;
				P1_Srobovanie.SkrutSet_K30.Cmd.ManualPresunBrzdu:= TRUE;
			ELSE
				P1_Srobovanie.SkrutSet_K30.Cmd.ManualPresunBrzdu:= FALSE;
			END_IF

			//Podanie skrutky//
			IF P1_Srobovanie.CMD.RR_SkrutSetK30_PodajSkrutku THEN
				P1_Srobovanie.CMD.RR_SkrutSetK30_PodajSkrutku:= FALSE;
				P1_Srobovanie.CMD.RR_SkrutSetK30_Zasobnik_RUN:= FALSE;
				P1_Srobovanie.SkrutSet_K30.Cmd.ManualStartHrniec:= FALSE;
				P1_Srobovanie.SkrutSet_K30.Cmd.ManualPresunBrzdu:= FALSE;
				P1_Srobovanie.CMD.PodajSkrutku_K30:= TRUE;
				SC_SkrutkovaciSet_K30.ResetStep:= TRUE;
				SC_SkrutkovaciSet_K30.Step:= 10;
			END_IF

	END_CASE

	//***********************************Skrutkovací set M4**************************************//
	//Volanie funkcie SequenceControl//
	SequenceControl(SC:= SC_SkrutkovaciSet_M4);

	CASE SC_SkrutkovaciSet_M4.Step OF

		0:
			SC_SkrutkovaciSet_M4.StepName:='0 - Nulovanie';
			P1_Srobovanie.SkrutSet_M4.CMD.ENABLE:= FALSE;
			P1_Srobovanie.SkrutSet_M4.CMD.RucnyRezim:= FALSE;
			P1_Srobovanie.SkrutSet_M4.CMD.PodajSkrutku:= FALSE;
			P1_Srobovanie.SkrutSet_M4.CMD.RR_OtocPodavac_Vstup:= FALSE;
			P1_Srobovanie.SkrutSet_M4.CMD.RR_OtocPodavac_Vystup:= FALSE;
			P1_Srobovanie.SkrutSet_M4.CMD.RR_ZapniVibrolistu:= FALSE;
			P1_Srobovanie.SkrutSet_M4.CMD.RR_ZapniZasobnik:= FALSE;

			IF SC_P1_Srobovanie.Step <> 0 THEN
				SC_SkrutkovaciSet_M4.ResetStep:= TRUE;
				SC_SkrutkovaciSet_M4.Step:= 1;
			END_IF

		1:
			SC_SkrutkovaciSet_M4.StepName:='1 - Rozhodnutie o cinnosti';

			IF P1_Srobovanie.Automat THEN
				SC_SkrutkovaciSet_M4.ResetStep:= TRUE;
				SC_SkrutkovaciSet_M4.Step:= 10;
			ELSIF P1_Srobovanie.Manual THEN
				SC_SkrutkovaciSet_M4.ResetStep:= TRUE;
				SC_SkrutkovaciSet_M4.Step:= 20;
			END_IF

		10:
			SC_SkrutkovaciSet_M4.StepName:='10 - Automaticky rezim - cakam na signal podaj skrutku';
			SC_SkrutkovaciSet_M4.IdleTime.PT:= T#2s;
			SC_SkrutkovaciSet_M4.AlarmTime.PT:= T#5s;

			P1_Srobovanie.SkrutSet_M4.CMD.ENABLE:= TRUE;

			IF P1_Srobovanie.CMD.PodajSkrutku_M4 THEN
				P1_Srobovanie.CMD.PodajSkrutku_M4:= FALSE;
				SC_SkrutkovaciSet_M4.ResetStep:= TRUE;
				SC_SkrutkovaciSet_M4.Step:= 13;
			END_IF

		13:
			SC_SkrutkovaciSet_M4.StepName:='13 - Automaticky rezim - podanie skrutky';
			SC_SkrutkovaciSet_M4.IdleTime.PT:= T#2s;
			SC_SkrutkovaciSet_M4.AlarmTime.PT:= T#5s;

			IF NOT SC_SkrutkovaciSet_M4.Switch1 THEN
				P1_Srobovanie.SkrutSet_M4.CMD.PodajSkrutku:= TRUE;
				SC_SkrutkovaciSet_M4.Switch1:= TRUE;
			END_IF

			IF P1_Srobovanie.SkrutSet_M4.STAV.SkrutkaPripravena THEN
				P1_Srobovanie.SkrutSet_M4.CMD.PodajSkrutku:= FALSE;
				SC_SkrutkovaciSet_M4.ResetStep:= TRUE;
				SC_SkrutkovaciSet_M4.Step:= 15;
			ELSIF P1_Srobovanie.SkrutSet_M4.STAV.ERROR THEN
				P1_Srobovanie.SkrutSet_M4.CMD.PodajSkrutku:= FALSE;
				P1_Alarmy[121]:= TRUE;
				P1_Pracovisko.STAV.Porucha_ST2:= TRUE;
			END_IF

		15:
			SC_SkrutkovaciSet_M4.StepName:='15 - Automaticky rezim - ukoncenie podania skrutky M4';
			SC_SkrutkovaciSet_M4.IdleTime.PT:= T#2s;
			SC_SkrutkovaciSet_M4.AlarmTime.PT:= T#5s;

			IF P1_Srobovanie.Manual THEN
				SC_SkrutkovaciSet_M4.ResetStep:= TRUE;
				SC_SkrutkovaciSet_M4.Step:= 20;
			ELSE
				SC_SkrutkovaciSet_M4.ResetStep:= TRUE;
				SC_SkrutkovaciSet_M4.Step:= 10;
			END_IF

		20:
			SC_SkrutkovaciSet_M4.StepName:='20 - Manualny rezim';
			SC_SkrutkovaciSet_M4.IdleTime.PT:= T#2s;
			SC_SkrutkovaciSet_M4.AlarmTime.PT:= T#5s;

			P1_Srobovanie.SkrutSet_M4.CMD.ENABLE:= TRUE;
			P1_Srobovanie.SkrutSet_M4.CMD.RucnyRezim:= TRUE;

			//Ovládanie zásobníka//
			IF P1_Srobovanie.CMD.RR_SkrutSetM4_Zasobnik_RUN THEN
				P1_Srobovanie.SkrutSet_M4.CMD.RR_ZapniZasobnik:= TRUE;
			ELSE
				P1_Srobovanie.SkrutSet_M4.CMD.RR_ZapniZasobnik:= FALSE;
			END_IF

			//Ovládanie vibrolišty//
			IF P1_Srobovanie.CMD.RR_SkrutSetM4_Vibrolista_RUN THEN
				P1_Srobovanie.SkrutSet_M4.CMD.RR_ZapniVibrolistu:= TRUE;
			ELSE
				P1_Srobovanie.SkrutSet_M4.CMD.RR_ZapniVibrolistu:= FALSE;
			END_IF

			//Otáčanie podavača skrutiek//
			IF P1_Srobovanie.CMD.RR_SkrutSetM4_OtocPodavac_Vstup THEN
				P1_Srobovanie.SkrutSet_M4.CMD.RR_OtocPodavac_Vstup:= TRUE;
				P1_Srobovanie.CMD.RR_SkrutSetM4_OtocPodavac_Vstup:= FALSE;
			ELSIF P1_Srobovanie.CMD.RR_SkrutSetM4_OtocPodavac_Vystup THEN
				P1_Srobovanie.SkrutSet_M4.CMD.RR_OtocPodavac_Vystup:= TRUE;
				P1_Srobovanie.CMD.RR_SkrutSetM4_OtocPodavac_Vystup:= FALSE;
			END_IF

			//Podanie skrutky//
			IF P1_Srobovanie.CMD.RR_SkrutSetM4_PodajSkrutku THEN
				P1_Srobovanie.CMD.RR_SkrutSetM4_PodajSkrutku:= FALSE;
				P1_Srobovanie.CMD.RR_SkrutSetM4_Zasobnik_RUN:= FALSE;
				P1_Srobovanie.CMD.RR_SkrutSetM4_Vibrolista_RUN:= FALSE;
				P1_Srobovanie.SkrutSet_M4.CMD.RucnyRezim:= TRUE;
				P1_Srobovanie.CMD.PodajSkrutku_M4:= TRUE;
				SC_SkrutkovaciSet_M4.ResetStep:= TRUE;
				SC_SkrutkovaciSet_M4.Step:= 10;
			END_IF

	END_CASE

	//***********************************Skrutkovací set M5***************************************//
	//Volanie funkcie SequenceControl//
	SequenceControl(SC:= SC_SkrutkovaciSet_M5);

	CASE SC_SkrutkovaciSet_M5.Step OF

		0:
			SC_SkrutkovaciSet_M5.StepName:='0 - Nulovanie';
			P1_Srobovanie.SkrutSet_M5.CMD.ENABLE:= FALSE;
			P1_Srobovanie.SkrutSet_M5.CMD.RucnyRezim:= FALSE;
			P1_Srobovanie.SkrutSet_M5.CMD.PodajSkrutku:= FALSE;
			P1_Srobovanie.SkrutSet_M5.CMD.RR_OtocPodavac_Vstup:= FALSE;
			P1_Srobovanie.SkrutSet_M5.CMD.RR_OtocPodavac_Vystup:= FALSE;
			P1_Srobovanie.SkrutSet_M5.CMD.RR_ZapniVibrolistu:= FALSE;
			P1_Srobovanie.SkrutSet_M5.CMD.RR_ZapniZasobnik:= FALSE;

			IF SC_P1_Srobovanie.Step <> 0 THEN
				SC_SkrutkovaciSet_M5.ResetStep:= TRUE;
				SC_SkrutkovaciSet_M5.Step:= 1;
			END_IF

		1:
			SC_SkrutkovaciSet_M5.StepName:='1 - Rozhodnutie o cinnosti';

			IF P1_Srobovanie.Automat THEN
				SC_SkrutkovaciSet_M5.ResetStep:= TRUE;
				SC_SkrutkovaciSet_M5.Step:= 10;
			ELSIF P1_Srobovanie.Manual THEN
				SC_SkrutkovaciSet_M5.ResetStep:= TRUE;
				SC_SkrutkovaciSet_M5.Step:= 20;
			END_IF

		10:
			SC_SkrutkovaciSet_M5.StepName:='10 - Automaticky rezim - cakam na signal podaj skrutku';
			SC_SkrutkovaciSet_M5.IdleTime.PT:= T#2s;
			SC_SkrutkovaciSet_M5.AlarmTime.PT:= T#5s;

			P1_Srobovanie.SkrutSet_M5.CMD.ENABLE:= TRUE;

			IF P1_Srobovanie.CMD.PodajSkrutku_M5 THEN
				P1_Srobovanie.CMD.PodajSkrutku_M5:= FALSE;
				SC_SkrutkovaciSet_M5.ResetStep:= TRUE;
				SC_SkrutkovaciSet_M5.Step:= 13;
			END_IF

		13:
			SC_SkrutkovaciSet_M5.StepName:='13 - Automaticky rezim - podanie skrutky';
			SC_SkrutkovaciSet_M5.IdleTime.PT:= T#2s;
			SC_SkrutkovaciSet_M5.AlarmTime.PT:= T#5s;

			IF NOT SC_SkrutkovaciSet_M5.Switch1 THEN
				P1_Srobovanie.SkrutSet_M5.CMD.PodajSkrutku:= TRUE;
				SC_SkrutkovaciSet_M5.Switch1:= TRUE;
			END_IF

			IF P1_Srobovanie.SkrutSet_M5.STAV.SkrutkaPripravena THEN
				P1_Srobovanie.SkrutSet_M5.CMD.PodajSkrutku:= FALSE;
				SC_SkrutkovaciSet_M5.ResetStep:= TRUE;
				SC_SkrutkovaciSet_M5.Step:= 15;
			ELSIF P1_Srobovanie.SkrutSet_M5.STAV.ERROR THEN
				P1_Srobovanie.SkrutSet_M5.CMD.PodajSkrutku:= FALSE;
				P1_Alarmy[120]:= TRUE;
				P1_Pracovisko.STAV.Porucha_ST2:= TRUE;
			END_IF

		15:
			SC_SkrutkovaciSet_M5.StepName:='15 - Automaticky rezim - ukoncenie podania skrutky M5';
			SC_SkrutkovaciSet_M5.IdleTime.PT:= T#2s;
			SC_SkrutkovaciSet_M5.AlarmTime.PT:= T#5s;

			IF P1_Srobovanie.Manual THEN
				SC_SkrutkovaciSet_M5.ResetStep:= TRUE;
				SC_SkrutkovaciSet_M5.Step:= 20;
			ELSE
				SC_SkrutkovaciSet_M5.ResetStep:= TRUE;
				SC_SkrutkovaciSet_M5.Step:= 10;
			END_IF

		20:
			SC_SkrutkovaciSet_M5.StepName:='20 - Manualny rezim';
			SC_SkrutkovaciSet_M5.IdleTime.PT:= T#2s;
			SC_SkrutkovaciSet_M5.AlarmTime.PT:= T#5s;

			P1_Srobovanie.SkrutSet_M5.CMD.ENABLE:= TRUE;
			P1_Srobovanie.SkrutSet_M5.CMD.RucnyRezim:= TRUE;

			//Ovládanie zásobníka//
			IF P1_Srobovanie.CMD.RR_SkrutSetM5_Zasobnik_RUN THEN
				P1_Srobovanie.SkrutSet_M5.CMD.RR_ZapniZasobnik:= TRUE;
			ELSE
				P1_Srobovanie.SkrutSet_M5.CMD.RR_ZapniZasobnik:= FALSE;
			END_IF

			//Ovládanie vibrolišty//
			IF P1_Srobovanie.CMD.RR_SkrutSetM5_Vibrolista_RUN THEN
				P1_Srobovanie.SkrutSet_M5.CMD.RR_ZapniVibrolistu:= TRUE;
			ELSE
				P1_Srobovanie.SkrutSet_M5.CMD.RR_ZapniVibrolistu:= FALSE;
			END_IF

			//Otáčanie podavača skrutiek//
			IF P1_Srobovanie.CMD.RR_SkrutSetM5_OtocPodavac_Vstup THEN
				P1_Srobovanie.SkrutSet_M5.CMD.RR_OtocPodavac_Vstup:= TRUE;
				P1_Srobovanie.CMD.RR_SkrutSetM5_OtocPodavac_Vstup:= FALSE;
			ELSIF P1_Srobovanie.CMD.RR_SkrutSetM5_OtocPodavac_Vystup THEN
				P1_Srobovanie.SkrutSet_M5.CMD.RR_OtocPodavac_Vystup:= TRUE;
				P1_Srobovanie.CMD.RR_SkrutSetM5_OtocPodavac_Vystup:= FALSE;
			END_IF

			//Podanie skrutky//
			IF P1_Srobovanie.CMD.RR_SkrutSetM5_PodajSkrutku THEN
				P1_Srobovanie.CMD.RR_SkrutSetM5_PodajSkrutku:= FALSE;
				P1_Srobovanie.CMD.RR_SkrutSetM5_Zasobnik_RUN:= FALSE;
				P1_Srobovanie.CMD.RR_SkrutSetM5_Vibrolista_RUN:= FALSE;
				P1_Srobovanie.SkrutSet_M5.CMD.RucnyRezim:= TRUE;
				P1_Srobovanie.CMD.PodajSkrutku_M5:= TRUE;
				SC_SkrutkovaciSet_M5.ResetStep:= TRUE;
				SC_SkrutkovaciSet_M5.Step:= 10;
			END_IF

	END_CASE

END_ACTION
```

### Program Logical/Program/Pracovisko_1/P1_Robot (IEC)

#### Main.st - Init, cyclic, exit code
```iecst
PROGRAM _INIT
	(* Insert code here *)

END_PROGRAM

PROGRAM _CYCLIC

	//Volanie funkcie SequenceControl//
	SequenceControl(SC:= SC_P1_Robot);

	//Volanie podprogramov//
	ProfinetKomunikaciaRobot;

	//Reset sekcie //
	IF P1_Robot.Reset THEN
		SC_P1_Robot.Step:= 0;
		P1_Robot.Reset:= FALSE;
	ELSIF NOT Safety.STAV.Linka_ZonaCS_AKTIVNA THEN
		SC_P1_Robot.Step:= 0;
	END_IF

	CASE SC_P1_Robot.Step OF

		0:
			SC_P1_Robot.StepName:='0 - Nulovanie';
			P1_Robot.Automat:= FALSE;
			P1_Robot.KoniecCyklu:= FALSE;
			P1_Robot.Manual:= FALSE;
			P1_Robot.Reset:= FALSE;
			P1_Robot.STAV.PoINIT:= FALSE;
			P1_Robot.COM_OUT.Odparkovanie:= FALSE;
			P1_Robot.COM_OUT.PP_na_Main:= FALSE;
			P1_Robot.COM_OUT.Reset_CS:= FALSE;
			P1_Robot.COM_OUT.StartProgramu:= FALSE;
			P1_Robot.COM_OUT.StartProgramuMain:= FALSE;
			P1_Robot.COM_OUT.VypniMotory:= FALSE;
			P1_Robot.COM_OUT.ZapniMotory:= FALSE;
			IF P1_Robot.COM_IN.Stav_RezimAUTOMAT AND P1_Robot.COM_IN.Stav_ProgramRUN THEN
				P1_Robot.COM_OUT.StopProgramu:= TRUE;
			ELSE
				P1_Robot.COM_OUT.StopProgramu:= FALSE;
			END_IF
			IF Safety.STAV.Linka_ZonaCS_AKTIVNA AND NOT P1_Pracovisko.STAV.Porucha_ST2 AND NOT P1_Robot.COM_IN.Stav_ProgramRUN AND P1_Pracovisko.STAV.HardwareBunky_OK THEN
				P1_Robot.COM_OUT.StopProgramu:= FALSE;
				SC_P1_Robot.ResetStep:= TRUE;
				SC_P1_Robot.Step:= 1;
			END_IF

		1:
			SC_P1_Robot.StepName:='1 - Cakam na spustenie vyroby';
			P1_Robot.KoniecCyklu:= FALSE;
			IF P1_Robot.Automat THEN
				SC_P1_Robot.Step:= 2;
			ELSIF P1_Robot.Manual THEN
				SC_P1_Robot.Step:= 700;
			END_IF

			//********************************************************Inicializácia****************************************************************************//

		2:
			SC_P1_Robot.StepName:='2 - Inicializacia - cakam na spustenie inicializacie';
			SC_P1_Robot.IdleTime.PT:= T#500ms;
			SC_P1_Robot.AlarmTime.PT:= T#5s;

			SC_P1_Robot.IdleTime.IN:= TRUE;

			P1_Robot.COM_OUT.VypniMotory:= TRUE;

			IF SC_P1_Robot.IdleTime.Q THEN
				SC_P1_Robot.ResetStep:= TRUE;
				SC_P1_Robot.Step:= 3;
			END_IF

		3:
			SC_P1_Robot.StepName:='2 - Inicializacia - kontrolujem central stop robota';
			SC_P1_Robot.IdleTime.PT:= T#500ms;
			SC_P1_Robot.AlarmTime.PT:= T#5s;

			IF P1_Robot.COM_IN.Stav_RobotCS THEN
				P1_Robot.COM_OUT.Reset_CS:= TRUE;
			END_IF

			IF NOT P1_Robot.COM_IN.Stav_RobotCS THEN
				P1_Robot.COM_OUT.Reset_CS:= FALSE;
				SC_P1_Robot.ResetStep:= TRUE;
				SC_P1_Robot.Step:= 4;
			END_IF

		4:
			SC_P1_Robot.StepName:='4 - Inicializacia - zapinam motory robota';
			SC_P1_Robot.IdleTime.PT:= T#500ms;
			SC_P1_Robot.AlarmTime.PT:= T#5s;

			IF NOT P1_Robot.COM_IN.Stav_MotoryON THEN
				P1_Robot.COM_OUT.VypniMotory:= FALSE;
				P1_Robot.COM_OUT.ZapniMotory:= TRUE;
			END_IF

			IF P1_Robot.COM_IN.Stav_MotoryON THEN
				P1_Robot.COM_OUT.ZapniMotory:= FALSE;
				SC_P1_Robot.ResetStep:= TRUE;
				SC_P1_Robot.Step:= 6;
			END_IF

		6:
			SC_P1_Robot.StepName:='6 - Inicializacia - spustam program robota od zaciatku';
			SC_P1_Robot.IdleTime.PT:= T#2s;
			SC_P1_Robot.AlarmTime.PT:= T#10s;

			SC_P1_Robot.IdleTime.IN:= P1_Robot.COM_IN.Stav_ProgramRUN;

			IF NOT SC_P1_Robot.Switch1 THEN
				P1_Robot.COM_OUT.StartProgramuMain:= TRUE;
				SC_P1_Robot.AlarmTime.IN:= TRUE;
				SC_P1_Robot.Switch1:= TRUE;
			END_IF

			IF SC_P1_Robot.IdleTime.Q AND P1_Robot.COM_IN.Stav_VystupyZresetovane THEN
				P1_Robot.COM_OUT.StartProgramuMain:= FALSE;
				P1_Robot.STAV.PoINIT:= TRUE;
				SC_P1_Robot.ResetStep:= TRUE;
				SC_P1_Robot.Step:= 100;
			ELSIF SC_P1_Robot.AlarmTime.Q THEN
				SC_P1_Robot.ResetStep:= TRUE;
				SC_P1_Robot.Step:= 0;
			END_IF

			//********************************************************Automatický režim****************************************************************************//

		100:
			SC_P1_Robot.StepName:='100 - Automaticky Rezim - cakam na ukoncenie programu robota';
			SC_P1_Robot.IdleTime.PT:= T#200ms;
			SC_P1_Robot.AlarmTime.PT:= T#5s;

			IF P1_Robot.KoniecCyklu AND NOT P1_StoperSrobovania.Automat AND NOT P1_Srobovanie.Automat AND P1_Robot.COM_IN.Stav_RobotOdparkovany THEN
				SC_P1_Robot.ResetStep:= TRUE;
				SC_P1_Robot.Step:= 0;
			ELSIF NOT P1_Robot.COM_IN.Stav_ProgramRUN THEN
				SC_P1_Robot.ResetStep:= TRUE;
				SC_P1_Robot.Step:= 0;
			END_IF

			//*******************************************************Manuálny režim*******************************************************************************//

		700:
			SC_P1_Robot.StepName:='700 - Manualny Rezim';
			SC_P1_Robot.IdleTime.PT:= T#8s;
			SC_P1_Robot.AlarmTime.PT:= T#5s;

	END_CASE

END_PROGRAM

PROGRAM _EXIT
	(* Insert code here *)

END_PROGRAM
```

#### ProfinetKomunikaciaRobot.st
```iecst
ACTION ProfinetKomunikaciaRobot:

	//Vstupy z Robota do PLC//
	P1_Robot.COM_IN.Stav_RezimAUTOMAT:= P1_Robot.COM_IN.BYTE_IN[0].0;
	P1_Robot.COM_IN.Stav_ProgramRUN:= P1_Robot.COM_IN.BYTE_IN[0].1;
	P1_Robot.COM_IN.Stav_MotoryOFF:= P1_Robot.COM_IN.BYTE_IN[0].2;
	P1_Robot.COM_IN.Stav_MotoryON:= P1_Robot.COM_IN.BYTE_IN[0].3;
	P1_Robot.COM_IN.Stav_RobotCS:= P1_Robot.COM_IN.BYTE_IN[0].4;

	P1_Robot.COM_IN.Stav_DPS_4F_Odobraty:= P1_Robot.COM_IN.BYTE_IN[1].0;
	P1_Robot.COM_IN.Stav_DPS_4F_Polozeny:= P1_Robot.COM_IN.BYTE_IN[1].1;
	P1_Robot.COM_IN.Stav_DPS_5F_Odobraty:= P1_Robot.COM_IN.BYTE_IN[1].2;
	P1_Robot.COM_IN.Stav_DPS_5F_Polozeny:= P1_Robot.COM_IN.BYTE_IN[1].3;
	P1_Robot.COM_IN.Stav_Foam4F_Odobraty:= P1_Robot.COM_IN.BYTE_IN[1].4;
	P1_Robot.COM_IN.Stav_Foam4F_Polozeny:= P1_Robot.COM_IN.BYTE_IN[1].5;
	P1_Robot.COM_IN.Stav_Foam5F_Odobraty:= P1_Robot.COM_IN.BYTE_IN[1].6;
	P1_Robot.COM_IN.Stav_Foam5F_Polozeny:= P1_Robot.COM_IN.BYTE_IN[1].7;

	P1_Robot.COM_IN.Stav_RobotBezpPozicia_Srobovanie:= TRUE;(*P1_Robot.COM_IN.BYTE_IN[2].0;*)
	P1_Robot.COM_IN.Stav_RobotOdparkovany:= P1_Robot.COM_IN.BYTE_IN[2].1;
	P1_Robot.COM_IN.Stav_RobotPoziciaCakania:= P1_Robot.COM_IN.BYTE_IN[2].2;
	P1_Robot.COM_IN.Stav_SpodnyBusbar4F_Odobraty:= P1_Robot.COM_IN.BYTE_IN[2].3;
	P1_Robot.COM_IN.Stav_SpodnyBusbar4F_Polozeny:= P1_Robot.COM_IN.BYTE_IN[2].4;
	P1_Robot.COM_IN.Stav_SpodnyBusbar5F_Odobraty:= P1_Robot.COM_IN.BYTE_IN[2].5;
	P1_Robot.COM_IN.Stav_SpodnyBusbar5F_Polozeny:= P1_Robot.COM_IN.BYTE_IN[2].6;
	P1_Robot.COM_IN.Stav_SpodnyBusbar5H_Odobraty:= P1_Robot.COM_IN.BYTE_IN[2].7;

	P1_Robot.COM_IN.Stav_SpodnyBusbar5H_Polozeny:= P1_Robot.COM_IN.BYTE_IN[3].0;
    P1_Robot.COM_IN.Stav_VystupyZresetovane:= P1_Robot.COM_IN.BYTE_IN[3].1;
    P1_Robot.COM_IN.Stav_BusbaryUvolnene:= P1_Robot.COM_IN.BYTE_IN[3].2;
    P1_Robot.COM_IN.Stav_RobotOdoberaBusbary:= P1_Robot.COM_IN.BYTE_IN[3].3;
    P1_Robot.COM_IN.Stav_RobotOdoberaFoamy:= P1_Robot.COM_IN.BYTE_IN[3].4;

	P1_Robot.OUT.OdistiGriper:= P1_Robot.COM_IN.BYTE_IN[4].0;
	P1_Robot.OUT.ZaistiGriper:= P1_Robot.COM_IN.BYTE_IN[4].1;
	P1_Robot.OUT.Griper_OTVOR:= P1_Robot.COM_IN.BYTE_IN[4].2;
	P1_Robot.OUT.Griper_ZATVOR:= P1_Robot.COM_IN.BYTE_IN[4].3;
	P1_Robot.OUT.Vakum_ON:= P1_Robot.COM_IN.BYTE_IN[4].4;
	P1_Robot.OUT.Vakum_OFF:= P1_Robot.COM_IN.BYTE_IN[4].5;

	//Vystupy z PLC do Robota//
	P1_Robot.COM_OUT.BYTE_OUT[0].0:= P1_Robot.COM_OUT.VypniMotory;
	P1_Robot.COM_OUT.BYTE_OUT[0].1:= P1_Robot.COM_OUT.ZapniMotory;
	P1_Robot.COM_OUT.BYTE_OUT[0].2:= P1_Robot.COM_OUT.PP_na_Main;
	P1_Robot.COM_OUT.BYTE_OUT[0].3:= P1_Robot.COM_OUT.StartProgramu;
	P1_Robot.COM_OUT.BYTE_OUT[0].4:= P1_Robot.COM_OUT.StartProgramuMain;
	P1_Robot.COM_OUT.BYTE_OUT[0].5:= P1_Robot.COM_OUT.StopProgramu;
	P1_Robot.COM_OUT.BYTE_OUT[0].6:= P1_Robot.COM_OUT.Reset_CS;

	P1_Robot.COM_OUT.BYTE_OUT[1].0:= P1_Robot.COM_OUT.ManipSrobovania_BezpecnaPozicia;
	P1_Robot.COM_OUT.BYTE_OUT[1].1:= P1_Robot.COM_OUT.OdoberDPS_4F_z_Paletky;
	P1_Robot.COM_OUT.BYTE_OUT[1].2:= P1_Robot.COM_OUT.OdoberDPS_5F_z_Paletky;
	P1_Robot.COM_OUT.BYTE_OUT[1].3:= P1_Robot.COM_OUT.OdoberFoam4F_z_Paletky;
	P1_Robot.COM_OUT.BYTE_OUT[1].4:= P1_Robot.COM_OUT.OdoberFoam5F_z_Paletky;
	P1_Robot.COM_OUT.BYTE_OUT[1].5:= P1_Robot.COM_OUT.OdoberSpodnyBusbar4F_z_Paletky;
	P1_Robot.COM_OUT.BYTE_OUT[1].6:= P1_Robot.COM_OUT.OdoberSpodnyBusbar5F_z_Paletky;
	P1_Robot.COM_OUT.BYTE_OUT[1].7:= P1_Robot.COM_OUT.OdoberSpodnyBusbar5H_z_Paletky;

	P1_Robot.COM_OUT.BYTE_OUT[2].0:= P1_Robot.COM_OUT.PolozDPS_4F_na_PowerCP;
	P1_Robot.COM_OUT.BYTE_OUT[2].1:= P1_Robot.COM_OUT.PolozDPS_5F_na_PowerCP;
	P1_Robot.COM_OUT.BYTE_OUT[2].2:= P1_Robot.COM_OUT.PolozFoam4F_na_PowerCP;
	P1_Robot.COM_OUT.BYTE_OUT[2].3:= P1_Robot.COM_OUT.PolozFoam5F_na_PowerCP;
	P1_Robot.COM_OUT.BYTE_OUT[2].4:= P1_Robot.COM_OUT.PolozSpodnyBusbar4F_na_PowerCP;
	P1_Robot.COM_OUT.BYTE_OUT[2].5:= P1_Robot.COM_OUT.PolozSpodnyBusbar5F_na_PowerCP;
	P1_Robot.COM_OUT.BYTE_OUT[2].6:= P1_Robot.COM_OUT.PolozSpodnyBusbar5H_na_PowerCP;
	P1_Robot.COM_OUT.BYTE_OUT[2].7:= P1_Robot.COM_OUT.Presun_CakaciaPozicia;

	P1_Robot.COM_OUT.BYTE_OUT[3].0:= P1_Robot.IN.DokStanica_PritomnGripra5H;
	P1_Robot.COM_OUT.BYTE_OUT[3].1:= P1_Robot.IN.DokStanica_PritomnGripra45F;
	P1_Robot.COM_OUT.BYTE_OUT[3].2:= P1_Robot.IN.Griper45F_Otvoreny;
	P1_Robot.COM_OUT.BYTE_OUT[3].3:= P1_Robot.IN.Griper45F_Zatvoreny;
	P1_Robot.COM_OUT.BYTE_OUT[3].4:= P1_Robot.IN.Vakum_OK;
	P1_Robot.COM_OUT.BYTE_OUT[3].5:= P1_Robot.IN.TypGripra_45F;
	P1_Robot.COM_OUT.BYTE_OUT[3].6:= P1_Robot.IN.TypGripra_5H;
    P1_Robot.COM_OUT.BYTE_OUT[3].7:= P1_Robot.COM_OUT.Odparkovanie;

    P1_Robot.COM_OUT.BYTE_OUT[4].0:= P1_Robot.COM_OUT.UvolniBusbary;
	P1_Robot.COM_OUT.BYTE_OUT[4].1:= P1_Robot.COM_OUT.ZopakujOdoberanie;

	//Typ gripra//
	P1_Robot.IN.TypGripra_45F:= P1_Robot.IN.KodGripra_Bit0 AND NOT P1_Robot.IN.KodGripra_Bit1;
	P1_Robot.IN.TypGripra_5H:= NOT P1_Robot.IN.KodGripra_Bit0 AND P1_Robot.IN.KodGripra_Bit1;

END_ACTION
```

### Program Logical/Program/Pracovisko_1/P1_AkumStoper (IEC)

#### Main.st - Init, cyclic, exit code
```iecst
PROGRAM _INIT
	(* Insert code here *)

END_PROGRAM

PROGRAM _CYCLIC

	//Volanie funkcie SequenceControl//
	SequenceControl(SC:= SC_P1_AkumulacnyStoper);

	//Reset sekcie //
	IF P1_AkumulacnyStoper.Reset THEN
		SC_P1_AkumulacnyStoper.Step:= 0;
		P1_AkumulacnyStoper.Reset:= FALSE;
	ELSIF NOT Safety.STAV.Linka_ZonaCS_AKTIVNA THEN
		SC_P1_AkumulacnyStoper.Step:= 0;
	END_IF

	CASE SC_P1_AkumulacnyStoper.Step OF

		0:
			SC_P1_AkumulacnyStoper.StepName:='0 - Nulovanie';
			P1_AkumulacnyStoper.Automat:= FALSE;
			P1_AkumulacnyStoper.KoniecCyklu:= FALSE;
			P1_AkumulacnyStoper.Manual:= FALSE;
			P1_AkumulacnyStoper.STAV.PoINIT:= FALSE;
			P1_AkumulacnyStoper.STAV.PrebiehaVyvezeniePaletky:= FALSE;
			P1_StoperSrobovania.STAV.PrebiehaVyvezeniePaletky:= FALSE;
			P1_AkumulacnyStoper.OUT.ZasunStoper:= FALSE;

			IF Safety.STAV.Linka_ZonaCS_AKTIVNA AND Safety.STAV.P1_ZonaBunky_AKTIVNA AND P1_Pracovisko.STAV.HardwareBunky_OK AND NOT P1_Pracovisko.STAV.Porucha_ST2 AND NOT P1_Pracovisko.STAV.Porucha_ST3 THEN
				SC_P1_AkumulacnyStoper.ResetStep:= TRUE;
				SC_P1_AkumulacnyStoper.Step:= 1;
			END_IF

		1:
			SC_P1_AkumulacnyStoper.StepName:='1 - Cakam na spustenie vyroby';
			P1_AkumulacnyStoper.KoniecCyklu:= FALSE;
			IF P1_AkumulacnyStoper.Automat THEN
				SC_P1_AkumulacnyStoper.Step:= 2;
			ELSIF P1_AkumulacnyStoper.Manual THEN
				SC_P1_AkumulacnyStoper.Step:= 700;
			END_IF

			//********************************************************Inicializácia****************************************************************************//
		2:
			SC_P1_AkumulacnyStoper.StepName:='2 - Inicializacia - cakam na spustenie inicializacie';
			SC_P1_AkumulacnyStoper.IdleTime.PT:= T#4s;
			SC_P1_AkumulacnyStoper.AlarmTime.PT:= T#5s;

			IF P1_Dopravniky.STAV.PoINIT THEN
				SC_P1_AkumulacnyStoper.ResetStep:= TRUE;
				SC_P1_AkumulacnyStoper.Step:= 3;
			END_IF

		3:
			SC_P1_AkumulacnyStoper.StepName:='3 - Inicializacia - hladanie paletky';
			SC_P1_AkumulacnyStoper.IdleTime.PT:= T#5s;
			SC_P1_AkumulacnyStoper.AlarmTime.PT:= T#5s;
			SC_P1_AkumulacnyStoper.IdleTime.IN:= TRUE;

			IF P1_AkumulacnyStoper.IN.PritomnostPaletky THEN
				P1_AkumulacnyStoper.STAV.PoINIT:= TRUE;
				SC_P1_AkumulacnyStoper.ResetStep:= TRUE;
				SC_P1_AkumulacnyStoper.Step:= 100;
			ELSIF SC_P1_AkumulacnyStoper.IdleTime.Q THEN
				P1_AkumulacnyStoper.STAV.PoINIT:= TRUE;
				SC_P1_AkumulacnyStoper.ResetStep:= TRUE;
				SC_P1_AkumulacnyStoper.Step:= 100;
			END_IF

			//********************************************************Automatický režim****************************************************************************//
		100:
			SC_P1_AkumulacnyStoper.StepName:='100 - Automaticky Rezim - cakam na príchod paletky na stoper';
			SC_P1_AkumulacnyStoper.IdleTime.PT:= T#200ms;
			SC_P1_AkumulacnyStoper.AlarmTime.PT:= T#5s;

			SC_P1_AkumulacnyStoper.IdleTime.IN:= P1_AkumulacnyStoper.IN.PritomnostPaletky;

			IF P1_AkumulacnyStoper.IN.PritomnostPaletky THEN
				P1_StoperSrobovania.STAV.PrebiehaVyvezeniePaletky:= FALSE;
			END_IF

			IF P1_AkumulacnyStoper.KoniecCyklu THEN
				SC_P1_AkumulacnyStoper.ResetStep:= TRUE;
				SC_P1_AkumulacnyStoper.Step:= 0;
			ELSIF SC_P1_AkumulacnyStoper.IdleTime.Q THEN
				SC_P1_AkumulacnyStoper.ResetStep:= TRUE;
				SC_P1_AkumulacnyStoper.Step:= 101;
			END_IF

		101:
			SC_P1_AkumulacnyStoper.StepName:='101 - Automaticky Rezim - cakam na vyvezenie paletky na stoper zakladania tesnenia';
			SC_P1_AkumulacnyStoper.IdleTime.PT:= T#200ms;
			SC_P1_AkumulacnyStoper.AlarmTime.PT:= T#5s;

			IF P1_AkumulacnyStoper.KoniecCyklu THEN
				SC_P1_AkumulacnyStoper.ResetStep:= TRUE;
				SC_P1_AkumulacnyStoper.Step:= 0;
			ELSIF SC_P2_StoperZaklTesnenia.Step = 100 AND NOT P2_StoperZaklTesnenia.RFID_hlava.PritomnostPaletky AND P2_ZakladacTesnenia.ServoPojazduZakladaca.Status.ActPosition < 10 AND NOT P1_AkumulacnyStoper.STAV.PrebiehaVyvezeniePaletky THEN
				SC_P1_AkumulacnyStoper.ResetStep:= TRUE;
				SC_P1_AkumulacnyStoper.Step:= 105;
			ELSIF NOT P1_AkumulacnyStoper.IN.PritomnostPaletky THEN
				SC_P1_AkumulacnyStoper.ResetStep:= TRUE;
				SC_P1_AkumulacnyStoper.Step:= 100;
			END_IF

		105:
			SC_P1_AkumulacnyStoper.StepName:='105 - Automaticky Rezim - vyvazam paletku na stoper zakladania tesnenia';
			SC_P1_AkumulacnyStoper.IdleTime.PT:= T#200ms;
			SC_P1_AkumulacnyStoper.AlarmTime.PT:= T#10s;

			SC_P1_AkumulacnyStoper.AlarmTime.IN:= P1_AkumulacnyStoper.IN.PritomnostPaletky;

			IF NOT SC_P1_AkumulacnyStoper.Switch1 THEN
				P1_AkumulacnyStoper.OUT.ZasunStoper:= TRUE;
				P1_AkumulacnyStoper.STAV.PrebiehaVyvezeniePaletky:= TRUE;
				SC_P1_AkumulacnyStoper.Switch1:= TRUE;
			END_IF

			IF NOT P1_AkumulacnyStoper.IN.PritomnostPaletky THEN
				P1_AkumulacnyStoper.OUT.ZasunStoper:= FALSE;
				SC_P1_AkumulacnyStoper.ResetStep:= TRUE;
				SC_P1_AkumulacnyStoper.Step:= 108;
			ELSIF SC_P1_AkumulacnyStoper.AlarmTime.Q THEN
				P1_Alarmy[162]:= TRUE;
				P1_Pracovisko.STAV.Porucha_ST3:= TRUE;
			END_IF

		108:
			SC_P1_AkumulacnyStoper.StepName:='108 - Automaticky Rezim - cakam na prichod paletky na stoper zakladania tesnenia';
			SC_P1_AkumulacnyStoper.IdleTime.PT:= T#200ms;
			SC_P1_AkumulacnyStoper.AlarmTime.PT:= T#10s;

			IF P2_StoperZaklTesnenia.RFID_hlava.PritomnostPaletky THEN
				P1_AkumulacnyStoper.STAV.PrebiehaVyvezeniePaletky:= FALSE;
				SC_P1_AkumulacnyStoper.ResetStep:= TRUE;
				SC_P1_AkumulacnyStoper.Step:= 100;
			END_IF

			//*******************************************************Manuálny režim*******************************************************************************//
		700:
			SC_P1_AkumulacnyStoper.StepName:='700 - Manualny Rezim';
			SC_P1_AkumulacnyStoper.IdleTime.PT:= T#8s;
			SC_P1_AkumulacnyStoper.AlarmTime.PT:= T#5s;

	END_CASE

END_PROGRAM

PROGRAM _EXIT
	(* Insert code here *)

END_PROGRAM
```

### Program Logical/Program/Pracovisko_1/P1_OvladVizu (IEC)
